(* CODESYS project elation_objectprog

Project tree, tasks and I/O mapping:
  Device : CODESYS Control for Linux SL, CODESYS, order no. 2302000005, version 4.13.0.0
    application Application
      libraries: Standard, 3.5.18.0 (System); Util, 3.5.19.0 (System); VisuDialogs, * (System)
      task MainTask (cyclic, interval t#4ms, priority 1) calls Main_program
      task VISU_TASK (cyclic, interval 100 ms, priority 31) calls VisuElems.Visu_Prg
      Chiller_funct/
        function maskbitFunction [ST]
        function scaleFunction [ST]
      function block clsLampFunction [ST]: Lamp, Switch, Value
      function block FB_Provision_room [ST]: MET_assign_values, P_Alarm, P_Defrost, P_Defrost_end_temperature, P_Door_open, P_Dout2, P_Dout3, P_Drain_down_time, P_Generic_alarm, P_High_temperature_alarm_threshold, P_High_temperature, P_Low_temperature, P_Low_temperature_alarm_threshold, P_Machine_standby, P_Maximum_defrost_duration, P_Provision_name, P_Room_temp, P_Setpoint, P_T1_failure, P_T2_failure, P_Temp_defrost, P_Thermostat_OFF_ON_ref_to_SP, P_Thermostat_ON_OFF_ref_to_SP, P_Time_based_defrost, MET_write_sepoint, P_setpoint_write, P_test_input, P_Thermostat_OFF_ON_ref_to_SP_write, P_Thermostat_ON_OFF_ref_to_SP_write, P_xTrigger_setpoint
      interface IProvroom: Lamp, Switch, Value
      interface ITF_provision_room: MET_assign_values, P_Alarm, P_Defrost, P_Defrost_end_temperature, P_Door_open, P_Dout2, P_Dout3, P_Drain_down_time, P_Generic_alarm, P_High_temperature, P_High_temperature_alarm_threshold, P_Low_temperature, P_Low_temperature_alarm_threshold, P_Machine_standby, P_Maximum_defrost_duration, P_Provision_name, P_Room_temp, P_Setpoint, P_T1_failure, P_T2_failure, P_Temp_defrost, P_Thermostat_OFF_ON_ref_to_SP, P_Thermostat_ON_OFF_ref_to_SP, P_Time_based_defrost, MET_write_sepoint, P_setpoint_write, P_test_input, P_Thermostat_OFF_ON_ref_to_SP_write, P_Thermostat_ON_OFF_ref_to_SP_write
      program Main_program [ST]
      visualisation MainVisualization
      visualisation objectvisiu
      visualisation Provision_1_2_3_SysOverview
      program Provision_1 [ST]
      visualisation Provision_1_Values
      program Provision_2 [ST]
      program Provision_3 [ST]
      program Provision_4 [ST]
      visualisation Provision_overview
      visualisation ProvRoom_All
      visualisation ProvRoomTemp
    Modbus_COM_2 : Modbus COM, CODESYS, version 4.4.0.0
        settings: ComPort = 2
      Modbus_Master_COM_Port : Modbus Client, COM Port, CODESYS, version 4.4.0.0
          settings: Auto-restart communication = TRUE
        Modbus_Slave_COM_Prov1 : Modbus Server, COM Port, CODESYS, version 4.4.0.0
            settings: Channel 0.Function Code = 3; Channel 0.Read Offset = 16#0000; Channel 0.Read Length = 18; Channel 0.Write Offset = 0; Channel 0.Write Length = 0; Channel 0.Cycle Time = 100; Channel 1.Function Code = 3; Channel 1.Read Offset = 16#0064; Channel 1.Read Length = 3; Channel 1.Write Offset = 0; Channel 1.Write Length = 0; Channel 1.Cycle Time = 100; Channel 2.Function Code = 3; Channel 2.Read Offset = 16#00C8; Channel 2.Read Length = 11; Channel 2.Write Offset = 0; Channel 2.Write Length = 0; Channel 2.Cycle Time = 100; Channel 3.Function Code = 3; Channel 3.Read Offset = 16#012C; Channel 3.Read Length = 10; Channel 3.Write Offset = 0; Channel 3.Write Length = 0; Channel 3.Cycle Time = 100; Channel 4.Function Code = 3; Channel 4.Read Offset = 16#0190; Channel 4.Read Length = 13; Channel 4.Write Offset = 0; Channel 4.Write Length = 0; Channel 4.Cycle Time = 100; Channel 5.Function Code = 3; Channel 5.Read Offset = 16#01F4; Channel 5.Read Length = 9; Channel 5.Write Offset = 0; Channel 5.Write Length = 0; Channel 5.Cycle Time = 100; Channel 6.Function Code = 3; Channel 6.Read Offset = 16#0258; Channel 6.Read Length = 10; Channel 6.Write Offset = 0;
              Channel 6.Write Length = 0; Channel 6.Cycle Time = 100; Channel 7.Function Code = 3; Channel 7.Read Offset = 16#02BE; Channel 7.Read Length = 2; Channel 7.Write Offset = 0; Channel 7.Write Length = 0; Channel 7.Cycle Time = 100; Channel 8.Function Code = 3; Channel 8.Read Offset = 16#01C2; Channel 8.Read Length = 8; Channel 8.Write Offset = 0; Channel 8.Write Length = 0; Channel 8.Cycle Time = 100; Channel 9.Function Code = 3; Channel 9.Read Offset = 16#00C1; Channel 9.Read Length = 5; Channel 9.Write Offset = 0; Channel 9.Write Length = 0; Channel 9.Cycle Time = 100; Channel 10.Function Code = 3; Channel 10.Read Offset = 16#028A; Channel 10.Read Length = 4; Channel 10.Write Offset = 0; Channel 10.Write Length = 0; Channel 10.Cycle Time = 100; Channel 11.Function Code = 6; Channel 11.Read Offset = 0; Channel 11.Read Length = 0; Channel 11.Write Offset = 16#012F; Channel 11.Write Length = 1; Channel 11.Cycle Time = 100; Channel 12.Function Code = 6; Channel 12.Read Offset = 0; Channel 12.Read Length = 0; Channel 12.Write Offset = 16#02BE; Channel 12.Write Length = 1; Channel 12.Cycle Time = 100; Channel 13.Function Code = 6; Channel 13.Read Offset = 0;
              Channel 13.Read Length = 0; Channel 13.Write Offset = 16#0130; Channel 13.Write Length = 1; Channel 13.Cycle Time = 100; Channel 14.Function Code = 6; Channel 14.Read Offset = 0; Channel 14.Read Length = 0; Channel 14.Write Offset = 16#0131; Channel 14.Write Length = 1; Channel 14.Cycle Time = 100; Channel 15.Function Code = 6; Channel 15.Read Offset = 0; Channel 15.Read Length = 0; Channel 15.Write Offset = 16#01F5; Channel 15.Write Length = 1; Channel 15.Cycle Time = 100; Channel 16.Function Code = 6; Channel 16.Read Offset = 0; Channel 16.Read Length = 0; Channel 16.Write Offset = 16#01F6; Channel 16.Write Length = 1; Channel 16.Cycle Time = 100; Channel 17.Function Code = 6; Channel 17.Read Offset = 0; Channel 17.Read Length = 0; Channel 17.Write Offset = 16#0079; Channel 17.Write Length = 1; Channel 17.Cycle Time = 100; Channel 18.Function Code = 6; Channel 18.Read Offset = 0; Channel 18.Read Length = 0; Channel 18.Write Offset = 16#0080; Channel 18.Write Length = 1; Channel 18.Cycle Time = 100; Channel 19.Function Code = 6; Channel 19.Read Offset = 0; Channel 19.Read Length = 0; Channel 19.Write Offset = 16#0191; Channel 19.Write Length = 1; Channel 19.Cycle Time = 100;
              Channel 20.Function Code = 6; Channel 20.Read Offset = 0; Channel 20.Read Length = 0; Channel 20.Write Offset = 16#0196; Channel 20.Write Length = 1; Channel 20.Cycle Time = 100; Channel 21.Function Code = 6; Channel 21.Read Offset = 0; Channel 21.Read Length = 0; Channel 21.Write Offset = 16#0198; Channel 21.Write Length = 1; Channel 21.Cycle Time = 100; Channel 22.Function Code = 6; Channel 22.Read Offset = 0; Channel 22.Read Length = 0; Channel 22.Write Offset = 16#0197; Channel 22.Write Length = 1; Channel 22.Cycle Time = 100; Channel 23.Function Code = 6; Channel 23.Read Offset = 0; Channel 23.Read Length = 0; Channel 23.Write Offset = 16#007A; Channel 23.Write Length = 1; Channel 23.Cycle Time = 100; Channel 24.Function Code = 6; Channel 24.Read Offset = 0; Channel 24.Read Length = 0; Channel 24.Write Offset = 16#01C2; Channel 24.Write Length = 1; Channel 24.Cycle Time = 100; Channel 25.Function Code = 6; Channel 25.Read Offset = 0; Channel 25.Read Length = 0; Channel 25.Write Offset = 16#00C8; Channel 25.Write Length = 1; Channel 25.Cycle Time = 100; Channel 26.Function Code = 6; Channel 26.Read Offset = 0; Channel 26.Read Length = 0; Channel 26.Write Offset = 16#012C;
              Channel 26.Write Length = 1; Channel 26.Cycle Time = 100; Channel 27.Function Code = 6; Channel 27.Read Offset = 0; Channel 27.Read Length = 0; Channel 27.Write Offset = 16#012D; Channel 27.Write Length = 1; Channel 27.Cycle Time = 100; Channel 28.Function Code = 6; Channel 28.Read Offset = 0; Channel 28.Read Length = 0; Channel 28.Write Offset = 16#012E; Channel 28.Write Length = 1; Channel 28.Cycle Time = 100; Channel 29.Function Code = 6; Channel 29.Read Offset = 0; Channel 29.Read Length = 0; Channel 29.Write Offset = 16#0132; Channel 29.Write Length = 1; Channel 29.Cycle Time = 100; Channel 30.Function Code = 6; Channel 30.Read Offset = 0; Channel 30.Read Length = 0; Channel 30.Write Offset = 16#0133; Channel 30.Write Length = 1; Channel 30.Cycle Time = 100; Channel 31.Function Code = 6; Channel 31.Read Offset = 0; Channel 31.Read Length = 0; Channel 31.Write Offset = 16#0134; Channel 31.Write Length = 1; Channel 31.Cycle Time = 100; Channel 32.Function Code = 6; Channel 32.Read Offset = 0; Channel 32.Read Length = 0; Channel 32.Write Offset = 16#0135; Channel 32.Write Length = 1; Channel 32.Cycle Time = 100; Channel 33.Function Code = 6; Channel 33.Read Offset = 0;
              Channel 33.Read Length = 0; Channel 33.Write Offset = 16#0192; Channel 33.Write Length = 1; Channel 33.Cycle Time = 100; Channel 34.Function Code = 6; Channel 34.Read Offset = 0; Channel 34.Read Length = 0; Channel 34.Write Offset = 16#0194; Channel 34.Write Length = 1; Channel 34.Cycle Time = 100; Channel 35.Function Code = 6; Channel 35.Read Offset = 0; Channel 35.Read Length = 0; Channel 35.Write Offset = 16#019C; Channel 35.Write Length = 1; Channel 35.Cycle Time = 100; Channel 36.Function Code = 6; Channel 36.Read Offset = 0; Channel 36.Read Length = 0; Channel 36.Write Offset = 16#019A; Channel 36.Write Length = 1; Channel 36.Cycle Time = 100; Channel 37.Function Code = 6; Channel 37.Read Offset = 0; Channel 37.Read Length = 0; Channel 37.Write Offset = 16#019B; Channel 37.Write Length = 1; Channel 37.Cycle Time = 100; Channel 45.Function Code = 6; Channel 45.Read Offset = 0; Channel 45.Read Length = 0; Channel 45.Write Offset = 16#01F4; Channel 45.Write Length = 1; Channel 45.Cycle Time = 100; Channel 39.Function Code = 6; Channel 39.Read Offset = 0; Channel 39.Read Length = 0; Channel 39.Write Offset = 16#01C3; Channel 39.Write Length = 1; Channel 39.Cycle Time = 100;
              Channel 40.Function Code = 6; Channel 40.Read Offset = 0; Channel 40.Read Length = 0; Channel 40.Write Offset = 16#01C4; Channel 40.Write Length = 1; Channel 40.Cycle Time = 100; Channel 41.Function Code = 6; Channel 41.Read Offset = 0; Channel 41.Read Length = 0; Channel 41.Write Offset = 16#01FA; Channel 41.Write Length = 1; Channel 41.Cycle Time = 100; Channel 42.Function Code = 6; Channel 42.Read Offset = 0; Channel 42.Read Length = 0; Channel 42.Write Offset = 16#0259; Channel 42.Write Length = 1; Channel 42.Cycle Time = 100; Channel 43.Function Code = 6; Channel 43.Read Offset = 0; Channel 43.Read Length = 0; Channel 43.Write Offset = 16#025A; Channel 43.Write Length = 1; Channel 43.Cycle Time = 100; Channel 44.Function Code = 6; Channel 44.Read Offset = 0; Channel 44.Read Length = 0; Channel 44.Write Offset = 16#025B; Channel 44.Write Length = 1; Channel 44.Cycle Time = 100; Channel 46.Function Code = 6; Channel 46.Read Offset = 0; Channel 46.Read Length = 0; Channel 46.Write Offset = 16#01F4; Channel 46.Write Length = 1; Channel 46.Cycle Time = 100; Channel 47.Function Code = 6; Channel 47.Read Offset = 0; Channel 47.Read Length = 0; Channel 47.Write Offset = 16#00D0;
              Channel 47.Write Length = 1; Channel 47.Cycle Time = 100; Channel 48.Function Code = 6; Channel 48.Read Offset = 0; Channel 48.Read Length = 0; Channel 48.Write Offset = 16#028A; Channel 48.Write Length = 1; Channel 48.Cycle Time = 100; Channel 49.Function Code = 6; Channel 49.Read Offset = 0; Channel 49.Read Length = 0; Channel 49.Write Offset = 16#028B; Channel 49.Write Length = 1; Channel 49.Cycle Time = 100; Channel 50.Function Code = 6; Channel 50.Read Offset = 0; Channel 50.Read Length = 0; Channel 50.Write Offset = 16#028C; Channel 50.Write Length = 1; Channel 50.Cycle Time = 100; Channel 51.Function Code = 6; Channel 51.Read Offset = 0; Channel 51.Read Length = 0; Channel 51.Write Offset = 16#028D; Channel 51.Write Length = 1; Channel 51.Cycle Time = 100; Channel 52.Function Code = 6; Channel 52.Read Offset = 0; Channel 52.Read Length = 0; Channel 52.Write Offset = 16#025C; Channel 52.Write Length = 1; Channel 52.Cycle Time = 100; Channel 53.Function Code = 6; Channel 53.Read Offset = 0; Channel 53.Read Length = 0; Channel 53.Write Offset = 16#025D; Channel 53.Write Length = 1; Channel 53.Cycle Time = 100; Channel 54.Function Code = 6; Channel 54.Read Offset = 0;
              Channel 54.Read Length = 0; Channel 54.Write Offset = 16#025E; Channel 54.Write Length = 1; Channel 54.Cycle Time = 100; Channel 55.Function Code = 6; Channel 55.Read Offset = 0; Channel 55.Read Length = 0; Channel 55.Write Offset = 16#025F; Channel 55.Write Length = 1; Channel 55.Cycle Time = 100; Channel 56.Function Code = 6; Channel 56.Read Offset = 0; Channel 56.Read Length = 0; Channel 56.Write Offset = 16#0260; Channel 56.Write Length = 1; Channel 56.Cycle Time = 100; Channel 57.Function Code = 6; Channel 57.Read Offset = 0; Channel 57.Read Length = 0; Channel 57.Write Offset = 16#0261; Channel 57.Write Length = 1; Channel 57.Cycle Time = 100; Channel 58.Function Code = 6; Channel 58.Read Offset = 0; Channel 58.Read Length = 0; Channel 58.Write Offset = 16#0193; Channel 58.Write Length = 1; Channel 58.Cycle Time = 100
            input  Application.Main_program.modbus_var[1,0] : WORD  // Channel 0.Channel 0
            input  Application.Main_program.modbus_var[1,1] : WORD  // Channel 0.Channel 0
            input  Application.Main_program.modbus_var[1,2] : WORD  // Channel 0.Channel 0
            input  Application.Main_program.modbus_var[1,3] : WORD  // Channel 0.Channel 0
            input  Application.Main_program.modbus_var[1,4] : WORD  // Channel 0.Channel 0
            input  Application.Main_program.modbus_var[1,5] : WORD  // Channel 0.Channel 0
            input  Application.Main_program.modbus_var[1,6] : WORD  // Channel 0.Channel 0
            input  Application.Main_program.modbus_var[1,7] : WORD  // Channel 0.Channel 0
            input  Application.Main_program.modbus_var[1,8] : WORD  // Channel 0.Channel 0
            input  Application.Main_program.modbus_var[1,9] : WORD  // Channel 0.Channel 0
            input  Application.Main_program.modbus_var[1,10] : WORD  // Channel 0.Channel 0
            input  Application.Main_program.modbus_var[1,11] : WORD  // Channel 0.Channel 0
            input  Application.Main_program.modbus_var[1,12] : WORD  // Channel 0.Channel 0
            input  Application.Main_program.modbus_var[1,13] : WORD  // Channel 0.Channel 0
            input  Application.Main_program.modbus_var[1,14] : WORD  // Channel 0.Channel 0
            input  Application.Main_program.modbus_var[1,15] : WORD  // Channel 0.Channel 0
            input  Application.Main_program.modbus_var[1,16] : WORD  // Channel 0.Channel 0
            input  Application.Main_program.modbus_var[1,17] : WORD  // Channel 0.Channel 0
            input  Application.Main_program.modbus_var[1,100] : WORD  // Channel 1.Channel 1
            input  Application.Main_program.modbus_var[1,101] : WORD  // Channel 1.Channel 1
            input  Application.Main_program.modbus_var[1,102] : WORD  // Channel 1.Channel 1
            output Application.Provision_1.get_param_trigger.Q : BIT  // Channel 2
            input  Application.Main_program.modbus_var[1,200] : WORD  // Channel 2.Channel 2
            input  Application.Main_program.modbus_var[1,201] : WORD  // Channel 2.Channel 2
            input  Application.Main_program.modbus_var[1,202] : WORD  // Channel 2.Channel 2
            input  Application.Main_program.modbus_var[1,203] : WORD  // Channel 2.Channel 2
            input  Application.Main_program.modbus_var[1,204] : WORD  // Channel 2.Channel 2
            input  Application.Main_program.modbus_var[1,205] : WORD  // Channel 2.Channel 2
            input  Application.Main_program.modbus_var[1,206] : WORD  // Channel 2.Channel 2
            input  Application.Main_program.modbus_var[1,207] : WORD  // Channel 2.Channel 2
            input  Application.Main_program.modbus_var[1,208] : WORD  // Channel 2.Channel 2
            input  Application.Main_program.modbus_var[1,209] : WORD  // Channel 2.Channel 2
            input  Application.Main_program.modbus_var[1,210] : WORD  // Channel 2.Channel 2
            input  Application.Main_program.modbus_var[1,300] : WORD  // Channel 3.Channel 3
            input  Application.Main_program.modbus_var[1,301] : WORD  // Channel 3.Channel 3
            input  Application.Main_program.modbus_var[1,302] : WORD  // Channel 3.Channel 3
            input  Application.Main_program.modbus_var[1,303] : WORD  // Channel 3.Channel 3
            input  Application.Main_program.modbus_var[1,304] : WORD  // Channel 3.Channel 3
            input  Application.Main_program.modbus_var[1,305] : WORD  // Channel 3.Channel 3
            input  Application.Main_program.modbus_var[1,306] : WORD  // Channel 3.Channel 3
            input  Application.Main_program.modbus_var[1,307] : WORD  // Channel 3.Channel 3
            input  Application.Main_program.modbus_var[1,308] : WORD  // Channel 3.Channel 3
            input  Application.Main_program.modbus_var[1,309] : WORD  // Channel 3.Channel 3
            input  Application.Main_program.modbus_var[1,400] : WORD  // Channel 4.Channel 4
            input  Application.Main_program.modbus_var[1,401] : WORD  // Channel 4.Channel 4
            input  Application.Main_program.modbus_var[1,402] : WORD  // Channel 4.Channel 4
            input  Application.Main_program.modbus_var[1,403] : WORD  // Channel 4.Channel 4
            input  Application.Main_program.modbus_var[1,404] : WORD  // Channel 4.Channel 4
            input  Application.Main_program.modbus_var[1,405] : WORD  // Channel 4.Channel 4
            input  Application.Main_program.modbus_var[1,406] : WORD  // Channel 4.Channel 4
            input  Application.Main_program.modbus_var[1,407] : WORD  // Channel 4.Channel 4
            input  Application.Main_program.modbus_var[1,408] : WORD  // Channel 4.Channel 4
            input  Application.Main_program.modbus_var[1,409] : WORD  // Channel 4.Channel 4
            input  Application.Main_program.modbus_var[1,410] : WORD  // Channel 4.Channel 4
            input  Application.Main_program.modbus_var[1,411] : WORD  // Channel 4.Channel 4
            input  Application.Main_program.modbus_var[1,412] : WORD  // Channel 4.Channel 4
            input  Application.Main_program.modbus_var[1,500] : WORD  // Channel 5.Channel 5
            input  Application.Main_program.modbus_var[1,501] : WORD  // Channel 5.Channel 5
            input  Application.Main_program.modbus_var[1,502] : WORD  // Channel 5.Channel 5
            input  Application.Main_program.modbus_var[1,503] : WORD  // Channel 5.Channel 5
            input  Application.Main_program.modbus_var[1,504] : WORD  // Channel 5.Channel 5
            input  Application.Main_program.modbus_var[1,505] : WORD  // Channel 5.Channel 5
            input  Application.Main_program.modbus_var[1,506] : WORD  // Channel 5.Channel 5
            input  Application.Main_program.modbus_var[1,507] : WORD  // Channel 5.Channel 5
            input  Application.Main_program.modbus_var[1,508] : WORD  // Channel 5.Channel 5
            output Application.Provision_1.get_param_trigger.Q : BIT  // Channel 6
            input  Application.Main_program.modbus_var[1,600] : WORD  // Channel 6.Channel 6
            input  Application.Main_program.modbus_var[1,601] : WORD  // Channel 6.Channel 6
            input  Application.Main_program.modbus_var[1,602] : WORD  // Channel 6.Channel 6
            input  Application.Main_program.modbus_var[1,603] : WORD  // Channel 6.Channel 6
            input  Application.Main_program.modbus_var[1,604] : WORD  // Channel 6.Channel 6
            input  Application.Main_program.modbus_var[1,605] : WORD  // Channel 6.Channel 6
            input  Application.Main_program.modbus_var[1,606] : WORD  // Channel 6.Channel 6
            input  Application.Main_program.modbus_var[1,607] : WORD  // Channel 6.Channel 6
            input  Application.Main_program.modbus_var[1,608] : WORD  // Channel 6.Channel 6
            input  Application.Main_program.modbus_var[1,609] : WORD  // Channel 6.Channel 6
            output Application.Provision_1.get_param_trigger.Q : BIT  // Channel 7
            input  Application.Main_program.modbus_var[1,702] : WORD  // Channel 7.Channel 7
            input  Application.Main_program.modbus_var[1,703] : WORD  // Channel 7.Channel 7
            output Application.Provision_1.get_param_trigger.Q : BIT  // Channel 8
            input  Application.Main_program.modbus_var[1,450] : WORD  // Channel 8.Channel 8
            input  Application.Main_program.modbus_var[1,451] : WORD  // Channel 8.Channel 8
            input  Application.Main_program.modbus_var[1,452] : WORD  // Channel 8.Channel 8
            input  Application.Main_program.modbus_var[1,453] : WORD  // Channel 8.Channel 8
            input  Application.Main_program.modbus_var[1,454] : WORD  // Channel 8.Channel 8
            input  Application.Main_program.modbus_var[1,455] : WORD  // Channel 8.Channel 8
            input  Application.Main_program.modbus_var[1,456] : WORD  // Channel 8.Channel 8
            input  Application.Main_program.modbus_var[1,457] : WORD  // Channel 8.Channel 8
            output Application.Provision_1.get_param_trigger.Q : BIT  // Channel 9
            output Application.Provision_1.get_param_trigger.Q : BIT  // Channel 10
            input  Application.Main_program.modbus_var[1,650] : WORD  // Channel 10.Channel 10
            input  Application.Main_program.modbus_var[1,651] : WORD  // Channel 10.Channel 10
            input  Application.Main_program.modbus_var[1,652] : WORD  // Channel 10.Channel 10
            input  Application.Main_program.modbus_var[1,653] : WORD  // Channel 10.Channel 10
            output Application.Provision_1.write_data_setp.Q : BIT  // Channel 11
            output Application.Provision_1.setp_write_word : WORD  // Channel 11.Channel 11
            output Application.Provision_1.write_data_control.Q : BIT  // Channel 12
            output Application.Provision_1.standby_write : WORD  // Channel 12.Channel 12
            output Application.Provision_1.write_data_setp.Q : BIT  // Channel 13
            output Application.Provision_1.Thermostat_OFF_ON_write_word : WORD  // Channel 13.Channel 13
            output Application.Provision_1.write_data_setp.Q : BIT  // Channel 14
            output Application.Provision_1.Thermostat_ON_OFF_write_word : WORD  // Channel 14.Channel 14
            output Application.Provision_1.write_data_alarm.Q : BIT  // Channel 15
            output Application.Provision_1.Low_temperature_alarm_thres_write_word : WORD  // Channel 15.Channel 15
            output Application.Provision_1.write_data_alarm.Q : BIT  // Channel 16
            output Application.Provision_1.High_temperature_alarm_thres_write_word : WORD  // Channel 16.Channel 16
            output Application.Provision_1.write_data_mute.Q : BIT  // Channel 17
            output Application.Provision_1.muteAlarm : WORD  // Channel 17.Channel 17
            output Application.Provision_1.Time_based_defrost_write_word : WORD  // Channel 18.Channel 18
            output Application.Provision_1.write_data_defrost.Q : BIT  // Channel 19
            output Application.Provision_1.Time_based_defrost_write_word : WORD  // Channel 19.Channel 19
            output Application.Provision_1.write_data_defrost.Q : BIT  // Channel 20
            output Application.Provision_1.Defrost_end_temperature_write_word : WORD  // Channel 20.Channel 20
            output Application.Provision_1.write_data_defrost.Q : BIT  // Channel 21
            output Application.Provision_1.Drain_down_time_write_int : WORD  // Channel 21.Channel 21
            output Application.Provision_1.write_data_defrost.Q : BIT  // Channel 22
            output Application.Provision_1.Maximum_defrost_duration_write_word : WORD  // Channel 22.Channel 22
            output Application.Provision_1.write_data_man_defrost.Q : BIT  // Channel 23
            output Application.Provision_1.defrost_write : WORD  // Channel 23.Channel 23
            output Application.Provision_1.set_param_trigger.Q : BIT  // Channel 24
            output Application.Provision_1.Fan_stop_temperature_write_word : WORD  // Channel 24.Channel 24
            output Application.Provision_1.preset_parameters_write_int : WORD  // Channel 25.Channel 25
            output Application.Provision_1.set_param_trigger.Q : BIT  // Channel 26
            output Application.Provision_1.Readout_scale_write_int : WORD  // Channel 26.Channel 26
            output Application.Provision_1.set_param_trigger.Q : BIT  // Channel 27
            output Application.Provision_1.Minimum_temperature_setpoint_write_int : WORD  // Channel 27.Channel 27
            output Application.Provision_1.set_param_trigger.Q : BIT  // Channel 28
            output Application.Provision_1.Maximum_temperature_setpoint_write_int : WORD  // Channel 28.Channel 28
            output Application.Provision_1.set_param_trigger.Q : BIT  // Channel 29
            output Application.Provision_1.CH_minimum_OFF_time_write_int : WORD  // Channel 29.Channel 29
            output Application.Provision_1.set_param_trigger.Q : BIT  // Channel 30
            output Application.Provision_1.CH_minimum_ON_time_write_int : WORD  // Channel 30.Channel 30
            output Application.Provision_1.set_param_trigger.Q : BIT  // Channel 31
            output Application.Provision_1.CH_output_ON_when_probe_T1_is_faulty_write_int : WORD  // Channel 31.Channel 31
            output Application.Provision_1.set_param_trigger.Q : BIT  // Channel 32
            output Application.Provision_1.CH_output_OFF_when_probe_T1_is_faulty_write_int : WORD  // Channel 32.Channel 32
            output Application.Provision_1.set_param_trigger.Q : BIT  // Channel 33
            output Application.Provision_1.Minimum_Time_Between_Defrost_write_int : WORD  // Channel 33.Channel 33
            output Application.Provision_1.set_param_trigger.Q : BIT  // Channel 34
            output Application.Provision_1.Defrost_type_write_int : WORD  // Channel 34.Channel 34
            output Application.Provision_1.set_param_trigger.Q : BIT  // Channel 35
            output Application.Provision_1.Fan_restart_temperature_after_defrost_write_int : WORD  // Channel 35.Channel 35
            output Application.Provision_1.set_param_trigger.Q : BIT  // Channel 36
            output Application.Provision_1.Display_delay_write_int : WORD  // Channel 36.Channel 36
            output Application.Provision_1.set_param_trigger.Q : BIT  // Channel 37
            output Application.Provision_1.Fans_active_during_defrost_write_int : WORD  // Channel 37.Channel 37
            output Application.Provision_1.set_param_trigger.Q : BIT  // Channel 39
            output Application.Provision_1.Maximum_fan_stop_for_FDD_FET_write_int : WORD  // Channel 39.Channel 39
            output Application.Provision_1.set_param_trigger.Q : BIT  // Channel 40
            output Application.Provision_1.Fan_mode_during_thermostatic_control_write_int : WORD  // Channel 40.Channel 40
            output Application.Provision_1.set_param_trigger.Q : BIT  // Channel 41
            output Application.Provision_1.Temperature_alarm_delay_write_int : WORD  // Channel 41.Channel 41
            output Application.Provision_1.set_param_trigger.Q : BIT  // Channel 42
            output Application.Provision_1.Door_switch_input_mode_write_int : WORD  // Channel 42.Channel 42
            output Application.Provision_1.set_param_trigger.Q : BIT  // Channel 43
            output Application.Provision_1.Door_alarm_delay_write_int : WORD  // Channel 43.Channel 43
            output Application.Provision_1.set_param_trigger.Q : BIT  // Channel 44
            output Application.Provision_1.Compressor_stop_delay_write_int : WORD  // Channel 44.Channel 44
            output Application.Provision_1.set_param_trigger.Q : BIT  // Channel 46
            output Application.Provision_1.Alarm_threshold_management_write_int : WORD  // Channel 46.Channel 46
            output Application.Provision_1.set_param_trigger.Q : BIT  // Channel 47
            output Application.Provision_1.Display_slowdown_write_int : WORD  // Channel 47.Channel 47
            output Application.Provision_1.set_param_trigger.Q : BIT  // Channel 48
            output Application.Provision_1.RL1_output_operation_write_int : WORD  // Channel 48.Channel 48
            output Application.Provision_1.set_param_trigger.Q : BIT  // Channel 49
            output Application.Provision_1.RL2_output_operation_write_int : WORD  // Channel 49.Channel 49
            output Application.Provision_1.set_param_trigger.Q : BIT  // Channel 50
            output Application.Provision_1.RL3_output_operation_write_int : WORD  // Channel 50.Channel 50
            output Application.Provision_1.set_param_trigger.Q : BIT  // Channel 51
            output Application.Provision_1.RL4_output_operation_write_int : WORD  // Channel 51.Channel 51
            output Application.Provision_1.Door_stop_timeout_write_int : WORD  // Channel 52.Channel 52
            output Application.Provision_1.set_param_trigger.Q : BIT  // Channel 53
            output Application.Provision_1.DI1_digital_input_operation_write_int : WORD  // Channel 53.Channel 53
            output Application.Provision_1.set_param_trigger.Q : BIT  // Channel 54
            output Application.Provision_1.DI1_digital_input_activation_write_int : WORD  // Channel 54.Channel 54
            output Application.Provision_1.set_param_trigger.Q : BIT  // Channel 55
            output Application.Provision_1.DI2_digital_input_operation_write_int : WORD  // Channel 55.Channel 55
            output Application.Provision_1.set_param_trigger.Q : BIT  // Channel 56
            output Application.Provision_1.DI2_digital_input_activation_write_int : WORD  // Channel 56.Channel 56
            output Application.Provision_1.set_param_trigger.Q : BIT  // Channel 57
            output Application.Provision_1.Light_control_mode_write_int : WORD  // Channel 57.Channel 57
            output Application.Provision_1.set_param_trigger.Q : BIT  // Channel 58
            output Application.Provision_1.Defrost_time_optimization_write_int : WORD  // Channel 58.Channel 58
            unmapped channels: Channel 0, Channel 1, Channel 2, Channel 3, Channel 4, Channel 5, Channel 6, Channel 7, Channel 8, Channel 9, Channel 10, Channel 11, Channel 12, Channel 13, Channel 14, Channel 15, Channel 16, Channel 17, Channel 18, Channel 18, Channel 19, Channel 20, Channel 21, Channel 22, Channel 23, Channel 24, Channel 25, Channel 25, Channel 26, Channel 27, Channel 28, Channel 29, Channel 30, Channel 31, Channel 32, Channel 33, Channel 34, Channel 35, Channel 36, Channel 37,
              Channel 38, Channel 45, Channel 39, Channel 40, Channel 41, Channel 42, Channel 43, Channel 44, Channel 46, Channel 47, Channel 48, Channel 49, Channel 50, Channel 51, Channel 52, Channel 53, Channel 54, Channel 55, Channel 56, Channel 57, Channel 58
        Modbus_Slave_COM_Prov2 : Modbus Server, COM Port, CODESYS, version 4.4.0.0
            settings: SlaveAddress = 2; ResponseTimeout = 1000; UseExtendedFunctionCodes = TRUE; Channel 0.Function Code = 3; Channel 0.Read Offset = 16#0000; Channel 0.Read Length = 18; Channel 0.Write Offset = 0; Channel 0.Write Length = 0; Channel 0.Cycle Time = 100; Channel 1.Function Code = 3; Channel 1.Read Offset = 16#0064; Channel 1.Read Length = 3; Channel 1.Write Offset = 0; Channel 1.Write Length = 0; Channel 1.Cycle Time = 100; Channel 2.Function Code = 3; Channel 2.Read Offset = 16#00C8; Channel 2.Read Length = 11; Channel 2.Write Offset = 0; Channel 2.Write Length = 0; Channel 2.Cycle Time = 100; Channel 3.Function Code = 3; Channel 3.Read Offset = 16#012C; Channel 3.Read Length = 10; Channel 3.Write Offset = 0; Channel 3.Write Length = 0; Channel 3.Cycle Time = 100; Channel 4.Function Code = 3; Channel 4.Read Offset = 16#0190; Channel 4.Read Length = 13; Channel 4.Write Offset = 0; Channel 4.Write Length = 0; Channel 4.Cycle Time = 100; Channel 5.Function Code = 3; Channel 5.Read Offset = 16#01F4; Channel 5.Read Length = 9; Channel 5.Write Offset = 0; Channel 5.Write Length = 0; Channel 5.Cycle Time = 100; Channel 6.Function Code = 3;
              Channel 6.Read Offset = 16#0258; Channel 6.Read Length = 10; Channel 6.Write Offset = 0; Channel 6.Write Length = 0; Channel 6.Cycle Time = 100; Channel 7.Function Code = 3; Channel 7.Read Offset = 16#02BE; Channel 7.Read Length = 2; Channel 7.Write Offset = 0; Channel 7.Write Length = 0; Channel 7.Cycle Time = 100; Channel 8.Function Code = 3; Channel 8.Read Offset = 16#01C2; Channel 8.Read Length = 8; Channel 8.Write Offset = 0; Channel 8.Write Length = 0; Channel 8.Cycle Time = 100; Channel 9.Function Code = 3; Channel 9.Read Offset = 16#00C1; Channel 9.Read Length = 5; Channel 9.Write Offset = 0; Channel 9.Write Length = 0; Channel 9.Cycle Time = 100; Channel 10.Function Code = 3; Channel 10.Read Offset = 16#028A; Channel 10.Read Length = 4; Channel 10.Write Offset = 0; Channel 10.Write Length = 0; Channel 10.Cycle Time = 100; Channel 11.Function Code = 6; Channel 11.Read Offset = 0; Channel 11.Read Length = 0; Channel 11.Write Offset = 16#012F; Channel 11.Write Length = 1; Channel 11.Cycle Time = 100; Channel 12.Function Code = 6; Channel 12.Read Offset = 0; Channel 12.Read Length = 0; Channel 12.Write Offset = 16#02BE; Channel 12.Write Length = 1;
              Channel 12.Cycle Time = 100; Channel 13.Function Code = 6; Channel 13.Read Offset = 0; Channel 13.Read Length = 0; Channel 13.Write Offset = 16#0130; Channel 13.Write Length = 1; Channel 13.Cycle Time = 100; Channel 14.Function Code = 6; Channel 14.Read Offset = 0; Channel 14.Read Length = 0; Channel 14.Write Offset = 16#0131; Channel 14.Write Length = 1; Channel 14.Cycle Time = 100; Channel 15.Function Code = 6; Channel 15.Read Offset = 0; Channel 15.Read Length = 0; Channel 15.Write Offset = 16#01F5; Channel 15.Write Length = 1; Channel 15.Cycle Time = 100; Channel 16.Function Code = 6; Channel 16.Read Offset = 0; Channel 16.Read Length = 0; Channel 16.Write Offset = 16#01F6; Channel 16.Write Length = 1; Channel 16.Cycle Time = 100; Channel 17.Function Code = 6; Channel 17.Read Offset = 0; Channel 17.Read Length = 0; Channel 17.Write Offset = 16#0079; Channel 17.Write Length = 1; Channel 17.Cycle Time = 100; Channel 18.Function Code = 6; Channel 18.Read Offset = 0; Channel 18.Read Length = 0; Channel 18.Write Offset = 16#0080; Channel 18.Write Length = 1; Channel 18.Cycle Time = 100; Channel 19.Function Code = 6; Channel 19.Read Offset = 0; Channel 19.Read Length = 0;
              Channel 19.Write Offset = 16#0191; Channel 19.Write Length = 1; Channel 19.Cycle Time = 100; Channel 20.Function Code = 6; Channel 20.Read Offset = 0; Channel 20.Read Length = 0; Channel 20.Write Offset = 16#0196; Channel 20.Write Length = 1; Channel 20.Cycle Time = 100; Channel 21.Function Code = 6; Channel 21.Read Offset = 0; Channel 21.Read Length = 0; Channel 21.Write Offset = 16#0198; Channel 21.Write Length = 1; Channel 21.Cycle Time = 100; Channel 22.Function Code = 6; Channel 22.Read Offset = 0; Channel 22.Read Length = 0; Channel 22.Write Offset = 16#0197; Channel 22.Write Length = 1; Channel 22.Cycle Time = 100; Channel 23.Function Code = 6; Channel 23.Read Offset = 0; Channel 23.Read Length = 0; Channel 23.Write Offset = 16#007A; Channel 23.Write Length = 1; Channel 23.Cycle Time = 100; Channel 24.Function Code = 6; Channel 24.Read Offset = 0; Channel 24.Read Length = 0; Channel 24.Write Offset = 16#01C2; Channel 24.Write Length = 1; Channel 24.Cycle Time = 100; Channel 25.Function Code = 6; Channel 25.Read Offset = 0; Channel 25.Read Length = 0; Channel 25.Write Offset = 16#00C8; Channel 25.Write Length = 1; Channel 25.Cycle Time = 100; Channel 26.Function Code = 6;
              Channel 26.Read Offset = 0; Channel 26.Read Length = 0; Channel 26.Write Offset = 16#012C; Channel 26.Write Length = 1; Channel 26.Cycle Time = 100; Channel 27.Function Code = 6; Channel 27.Read Offset = 0; Channel 27.Read Length = 0; Channel 27.Write Offset = 16#012D; Channel 27.Write Length = 1; Channel 27.Cycle Time = 100; Channel 28.Function Code = 6; Channel 28.Read Offset = 0; Channel 28.Read Length = 0; Channel 28.Write Offset = 16#012E; Channel 28.Write Length = 1; Channel 28.Cycle Time = 100; Channel 29.Function Code = 6; Channel 29.Read Offset = 0; Channel 29.Read Length = 0; Channel 29.Write Offset = 16#0132; Channel 29.Write Length = 1; Channel 29.Cycle Time = 100; Channel 30.Function Code = 6; Channel 30.Read Offset = 0; Channel 30.Read Length = 0; Channel 30.Write Offset = 16#0133; Channel 30.Write Length = 1; Channel 30.Cycle Time = 100; Channel 31.Function Code = 6; Channel 31.Read Offset = 0; Channel 31.Read Length = 0; Channel 31.Write Offset = 16#0134; Channel 31.Write Length = 1; Channel 31.Cycle Time = 100; Channel 32.Function Code = 6; Channel 32.Read Offset = 0; Channel 32.Read Length = 0; Channel 32.Write Offset = 16#0135; Channel 32.Write Length = 1;
              Channel 32.Cycle Time = 100; Channel 33.Function Code = 6; Channel 33.Read Offset = 0; Channel 33.Read Length = 0; Channel 33.Write Offset = 16#0192; Channel 33.Write Length = 1; Channel 33.Cycle Time = 100; Channel 34.Function Code = 6; Channel 34.Read Offset = 0; Channel 34.Read Length = 0; Channel 34.Write Offset = 16#0194; Channel 34.Write Length = 1; Channel 34.Cycle Time = 100; Channel 35.Function Code = 6; Channel 35.Read Offset = 0; Channel 35.Read Length = 0; Channel 35.Write Offset = 16#019C; Channel 35.Write Length = 1; Channel 35.Cycle Time = 100; Channel 36.Function Code = 6; Channel 36.Read Offset = 0; Channel 36.Read Length = 0; Channel 36.Write Offset = 16#019A; Channel 36.Write Length = 1; Channel 36.Cycle Time = 100; Channel 37.Function Code = 6; Channel 37.Read Offset = 0; Channel 37.Read Length = 0; Channel 37.Write Offset = 16#019B; Channel 37.Write Length = 1; Channel 37.Cycle Time = 100; Channel 45.Function Code = 6; Channel 45.Read Offset = 0; Channel 45.Read Length = 0; Channel 45.Write Offset = 16#01F4; Channel 45.Write Length = 1; Channel 45.Cycle Time = 100; Channel 39.Function Code = 6; Channel 39.Read Offset = 0; Channel 39.Read Length = 0;
              Channel 39.Write Offset = 16#01C3; Channel 39.Write Length = 1; Channel 39.Cycle Time = 100; Channel 40.Function Code = 6; Channel 40.Read Offset = 0; Channel 40.Read Length = 0; Channel 40.Write Offset = 16#01C4; Channel 40.Write Length = 1; Channel 40.Cycle Time = 100; Channel 41.Function Code = 6; Channel 41.Read Offset = 0; Channel 41.Read Length = 0; Channel 41.Write Offset = 16#01FA; Channel 41.Write Length = 1; Channel 41.Cycle Time = 100; Channel 42.Function Code = 6; Channel 42.Read Offset = 0; Channel 42.Read Length = 0; Channel 42.Write Offset = 16#0259; Channel 42.Write Length = 1; Channel 42.Cycle Time = 100; Channel 43.Function Code = 6; Channel 43.Read Offset = 0; Channel 43.Read Length = 0; Channel 43.Write Offset = 16#025A; Channel 43.Write Length = 1; Channel 43.Cycle Time = 100; Channel 44.Function Code = 6; Channel 44.Read Offset = 0; Channel 44.Read Length = 0; Channel 44.Write Offset = 16#025B; Channel 44.Write Length = 1; Channel 44.Cycle Time = 100; Channel 46.Function Code = 6; Channel 46.Read Offset = 0; Channel 46.Read Length = 0; Channel 46.Write Offset = 16#01F4; Channel 46.Write Length = 1; Channel 46.Cycle Time = 100; Channel 47.Function Code = 6;
              Channel 47.Read Offset = 0; Channel 47.Read Length = 0; Channel 47.Write Offset = 16#00D0; Channel 47.Write Length = 1; Channel 47.Cycle Time = 100; Channel 48.Function Code = 6; Channel 48.Read Offset = 0; Channel 48.Read Length = 0; Channel 48.Write Offset = 16#028A; Channel 48.Write Length = 1; Channel 48.Cycle Time = 100; Channel 49.Function Code = 6; Channel 49.Read Offset = 0; Channel 49.Read Length = 0; Channel 49.Write Offset = 16#028B; Channel 49.Write Length = 1; Channel 49.Cycle Time = 100; Channel 50.Function Code = 6; Channel 50.Read Offset = 0; Channel 50.Read Length = 0; Channel 50.Write Offset = 16#028C; Channel 50.Write Length = 1; Channel 50.Cycle Time = 100; Channel 51.Function Code = 6; Channel 51.Read Offset = 0; Channel 51.Read Length = 0; Channel 51.Write Offset = 16#028D; Channel 51.Write Length = 1; Channel 51.Cycle Time = 100; Channel 52.Function Code = 6; Channel 52.Read Offset = 0; Channel 52.Read Length = 0; Channel 52.Write Offset = 16#025C; Channel 52.Write Length = 1; Channel 52.Cycle Time = 100; Channel 53.Function Code = 6; Channel 53.Read Offset = 0; Channel 53.Read Length = 0; Channel 53.Write Offset = 16#025D; Channel 53.Write Length = 1;
              Channel 53.Cycle Time = 100; Channel 54.Function Code = 6; Channel 54.Read Offset = 0; Channel 54.Read Length = 0; Channel 54.Write Offset = 16#025E; Channel 54.Write Length = 1; Channel 54.Cycle Time = 100; Channel 55.Function Code = 6; Channel 55.Read Offset = 0; Channel 55.Read Length = 0; Channel 55.Write Offset = 16#025F; Channel 55.Write Length = 1; Channel 55.Cycle Time = 100; Channel 56.Function Code = 6; Channel 56.Read Offset = 0; Channel 56.Read Length = 0; Channel 56.Write Offset = 16#0260; Channel 56.Write Length = 1; Channel 56.Cycle Time = 100; Channel 57.Function Code = 6; Channel 57.Read Offset = 0; Channel 57.Read Length = 0; Channel 57.Write Offset = 16#0261; Channel 57.Write Length = 1; Channel 57.Cycle Time = 100; Channel 58.Function Code = 6; Channel 58.Read Offset = 0; Channel 58.Read Length = 0; Channel 58.Write Offset = 16#0193; Channel 58.Write Length = 1; Channel 58.Cycle Time = 100
            input  Application.Main_program.modbus_var[2,0] : WORD  // Channel 0.Channel 0
            input  Application.Main_program.modbus_var[2,1] : WORD  // Channel 0.Channel 0
            input  Application.Main_program.modbus_var[2,2] : WORD  // Channel 0.Channel 0
            input  Application.Main_program.modbus_var[2,3] : WORD  // Channel 0.Channel 0
            input  Application.Main_program.modbus_var[2,4] : WORD  // Channel 0.Channel 0
            input  Application.Main_program.modbus_var[2,5] : WORD  // Channel 0.Channel 0
            input  Application.Main_program.modbus_var[2,6] : WORD  // Channel 0.Channel 0
            input  Application.Main_program.modbus_var[2,7] : WORD  // Channel 0.Channel 0
            input  Application.Main_program.modbus_var[2,8] : WORD  // Channel 0.Channel 0
            input  Application.Main_program.modbus_var[2,9] : WORD  // Channel 0.Channel 0
            input  Application.Main_program.modbus_var[2,10] : WORD  // Channel 0.Channel 0
            input  Application.Main_program.modbus_var[2,11] : WORD  // Channel 0.Channel 0
            input  Application.Main_program.modbus_var[2,12] : WORD  // Channel 0.Channel 0
            input  Application.Main_program.modbus_var[2,13] : WORD  // Channel 0.Channel 0
            input  Application.Main_program.modbus_var[2,14] : WORD  // Channel 0.Channel 0
            input  Application.Main_program.modbus_var[2,15] : WORD  // Channel 0.Channel 0
            input  Application.Main_program.modbus_var[2,16] : WORD  // Channel 0.Channel 0
            input  Application.Main_program.modbus_var[2,17] : WORD  // Channel 0.Channel 0
            input  Application.Main_program.modbus_var[2,100] : WORD  // Channel 1.Channel 1
            input  Application.Main_program.modbus_var[2,101] : WORD  // Channel 1.Channel 1
            input  Application.Main_program.modbus_var[2,102] : WORD  // Channel 1.Channel 1
            output Application.Provision_2.get_param_trigger.Q : BIT  // Channel 2
            input  Application.Main_program.modbus_var[2,200] : WORD  // Channel 2.Channel 2
            input  Application.Main_program.modbus_var[2,201] : WORD  // Channel 2.Channel 2
            input  Application.Main_program.modbus_var[2,202] : WORD  // Channel 2.Channel 2
            input  Application.Main_program.modbus_var[2,203] : WORD  // Channel 2.Channel 2
            input  Application.Main_program.modbus_var[2,204] : WORD  // Channel 2.Channel 2
            input  Application.Main_program.modbus_var[2,205] : WORD  // Channel 2.Channel 2
            input  Application.Main_program.modbus_var[2,206] : WORD  // Channel 2.Channel 2
            input  Application.Main_program.modbus_var[2,207] : WORD  // Channel 2.Channel 2
            input  Application.Main_program.modbus_var[2,208] : WORD  // Channel 2.Channel 2
            input  Application.Main_program.modbus_var[2,209] : WORD  // Channel 2.Channel 2
            input  Application.Main_program.modbus_var[2,210] : WORD  // Channel 2.Channel 2
            input  Application.Main_program.modbus_var[2,300] : WORD  // Channel 3.Channel 3
            input  Application.Main_program.modbus_var[2,301] : WORD  // Channel 3.Channel 3
            input  Application.Main_program.modbus_var[2,302] : WORD  // Channel 3.Channel 3
            input  Application.Main_program.modbus_var[2,303] : WORD  // Channel 3.Channel 3
            input  Application.Main_program.modbus_var[2,304] : WORD  // Channel 3.Channel 3
            input  Application.Main_program.modbus_var[2,305] : WORD  // Channel 3.Channel 3
            input  Application.Main_program.modbus_var[2,306] : WORD  // Channel 3.Channel 3
            input  Application.Main_program.modbus_var[2,307] : WORD  // Channel 3.Channel 3
            input  Application.Main_program.modbus_var[2,308] : WORD  // Channel 3.Channel 3
            input  Application.Main_program.modbus_var[2,309] : WORD  // Channel 3.Channel 3
            input  Application.Main_program.modbus_var[2,400] : WORD  // Channel 4.Channel 4
            input  Application.Main_program.modbus_var[2,401] : WORD  // Channel 4.Channel 4
            input  Application.Main_program.modbus_var[2,402] : WORD  // Channel 4.Channel 4
            input  Application.Main_program.modbus_var[2,403] : WORD  // Channel 4.Channel 4
            input  Application.Main_program.modbus_var[2,404] : WORD  // Channel 4.Channel 4
            input  Application.Main_program.modbus_var[2,405] : WORD  // Channel 4.Channel 4
            input  Application.Main_program.modbus_var[2,406] : WORD  // Channel 4.Channel 4
            input  Application.Main_program.modbus_var[2,407] : WORD  // Channel 4.Channel 4
            input  Application.Main_program.modbus_var[2,408] : WORD  // Channel 4.Channel 4
            input  Application.Main_program.modbus_var[2,409] : WORD  // Channel 4.Channel 4
            input  Application.Main_program.modbus_var[2,410] : WORD  // Channel 4.Channel 4
            input  Application.Main_program.modbus_var[2,411] : WORD  // Channel 4.Channel 4
            input  Application.Main_program.modbus_var[2,412] : WORD  // Channel 4.Channel 4
            input  Application.Main_program.modbus_var[2,500] : WORD  // Channel 5.Channel 5
            input  Application.Main_program.modbus_var[2,501] : WORD  // Channel 5.Channel 5
            input  Application.Main_program.modbus_var[2,502] : WORD  // Channel 5.Channel 5
            input  Application.Main_program.modbus_var[2,503] : WORD  // Channel 5.Channel 5
            input  Application.Main_program.modbus_var[2,504] : WORD  // Channel 5.Channel 5
            input  Application.Main_program.modbus_var[2,505] : WORD  // Channel 5.Channel 5
            input  Application.Main_program.modbus_var[2,506] : WORD  // Channel 5.Channel 5
            input  Application.Main_program.modbus_var[2,507] : WORD  // Channel 5.Channel 5
            input  Application.Main_program.modbus_var[2,508] : WORD  // Channel 5.Channel 5
            output Application.Provision_2.get_param_trigger.Q : BIT  // Channel 6
            input  Application.Main_program.modbus_var[2,600] : WORD  // Channel 6.Channel 6
            input  Application.Main_program.modbus_var[2,601] : WORD  // Channel 6.Channel 6
            input  Application.Main_program.modbus_var[2,602] : WORD  // Channel 6.Channel 6
            input  Application.Main_program.modbus_var[2,603] : WORD  // Channel 6.Channel 6
            input  Application.Main_program.modbus_var[2,604] : WORD  // Channel 6.Channel 6
            input  Application.Main_program.modbus_var[2,605] : WORD  // Channel 6.Channel 6
            input  Application.Main_program.modbus_var[2,606] : WORD  // Channel 6.Channel 6
            input  Application.Main_program.modbus_var[2,607] : WORD  // Channel 6.Channel 6
            input  Application.Main_program.modbus_var[2,608] : WORD  // Channel 6.Channel 6
            input  Application.Main_program.modbus_var[2,609] : WORD  // Channel 6.Channel 6
            output Application.Provision_2.get_param_trigger.Q : BIT  // Channel 7
            input  Application.Main_program.modbus_var[2,702] : WORD  // Channel 7.Channel 7
            input  Application.Main_program.modbus_var[2,703] : WORD  // Channel 7.Channel 7
            output Application.Provision_2.get_param_trigger.Q : BIT  // Channel 8
            input  Application.Main_program.modbus_var[2,450] : WORD  // Channel 8.Channel 8
            input  Application.Main_program.modbus_var[2,451] : WORD  // Channel 8.Channel 8
            input  Application.Main_program.modbus_var[2,452] : WORD  // Channel 8.Channel 8
            input  Application.Main_program.modbus_var[2,453] : WORD  // Channel 8.Channel 8
            input  Application.Main_program.modbus_var[2,454] : WORD  // Channel 8.Channel 8
            input  Application.Main_program.modbus_var[2,455] : WORD  // Channel 8.Channel 8
            input  Application.Main_program.modbus_var[2,456] : WORD  // Channel 8.Channel 8
            input  Application.Main_program.modbus_var[2,457] : WORD  // Channel 8.Channel 8
            output Application.Provision_2.get_param_trigger.Q : BIT  // Channel 9
            output Application.Provision_2.get_param_trigger.Q : BIT  // Channel 10
            input  Application.Main_program.modbus_var[2,650] : WORD  // Channel 10.Channel 10
            input  Application.Main_program.modbus_var[2,651] : WORD  // Channel 10.Channel 10
            input  Application.Main_program.modbus_var[2,652] : WORD  // Channel 10.Channel 10
            input  Application.Main_program.modbus_var[2,653] : WORD  // Channel 10.Channel 10
            output Application.Main_program.Provision_room2.O_write_data_setp.Q : BIT  // Channel 11
            output Application.Main_program.Provision_room2.O_word_setpoint : WORD  // Channel 11.Channel 11
            output Application.Provision_2.write_data_control.Q : BIT  // Channel 12
            output Application.Provision_2.standby_write : WORD  // Channel 12.Channel 12
            output Application.Main_program.Provision_room2.O_write_data_setp.Q : BIT  // Channel 13
            output Application.Provision_2.Thermostat_OFF_ON_write_word : WORD  // Channel 13.Channel 13
            output Application.Main_program.Provision_room2.O_write_data_setp.Q : BIT  // Channel 14
            output Application.Provision_2.Thermostat_ON_OFF_write_word : WORD  // Channel 14.Channel 14
            output Application.Provision_2.write_data_alarm.Q : BIT  // Channel 15
            output Application.Provision_2.Low_temperature_alarm_thres_write_word : WORD  // Channel 15.Channel 15
            output Application.Provision_2.write_data_alarm.Q : BIT  // Channel 16
            output Application.Provision_2.High_temperature_alarm_thres_write_word : WORD  // Channel 16.Channel 16
            output Application.Provision_2.write_data_mute.Q : BIT  // Channel 17
            output Application.Provision_2.muteAlarm : WORD  // Channel 17.Channel 17
            output Application.Provision_2.Time_based_defrost_write_word : WORD  // Channel 18.Channel 18
            output Application.Provision_2.write_data_defrost.Q : BIT  // Channel 19
            output Application.Provision_2.Time_based_defrost_write_word : WORD  // Channel 19.Channel 19
            output Application.Provision_2.write_data_defrost.Q : BIT  // Channel 20
            output Application.Provision_2.Defrost_end_temperature_write_word : WORD  // Channel 20.Channel 20
            output Application.Provision_2.write_data_defrost.Q : BIT  // Channel 21
            output Application.Provision_2.Drain_down_time_write_int : WORD  // Channel 21.Channel 21
            output Application.Provision_2.write_data_defrost.Q : BIT  // Channel 22
            output Application.Provision_2.Maximum_defrost_duration_write_word : WORD  // Channel 22.Channel 22
            output Application.Provision_2.write_data_man_defrost.Q : BIT  // Channel 23
            output Application.Provision_2.defrost_write : WORD  // Channel 23.Channel 23
            output Application.Provision_2.set_param_trigger.Q : BIT  // Channel 24
            output Application.Provision_2.Fan_stop_temperature_write_word : WORD  // Channel 24.Channel 24
            output Application.Provision_2.preset_parameters_write_int : WORD  // Channel 25.Channel 25
            output Application.Provision_2.set_param_trigger.Q : BIT  // Channel 26
            output Application.Provision_2.Readout_scale_write_int : WORD  // Channel 26.Channel 26
            output Application.Provision_2.set_param_trigger.Q : BIT  // Channel 27
            output Application.Provision_2.Minimum_temperature_setpoint_write_int : WORD  // Channel 27.Channel 27
            output Application.Provision_2.set_param_trigger.Q : BIT  // Channel 28
            output Application.Provision_2.Maximum_temperature_setpoint_write_int : WORD  // Channel 28.Channel 28
            output Application.Provision_2.set_param_trigger.Q : BIT  // Channel 29
            output Application.Provision_2.CH_minimum_OFF_time_write_int : WORD  // Channel 29.Channel 29
            output Application.Provision_2.set_param_trigger.Q : BIT  // Channel 30
            output Application.Provision_2.CH_minimum_ON_time_write_int : WORD  // Channel 30.Channel 30
            output Application.Provision_2.set_param_trigger.Q : BIT  // Channel 31
            output Application.Provision_2.CH_output_ON_when_probe_T1_is_faulty_write_int : WORD  // Channel 31.Channel 31
            output Application.Provision_2.set_param_trigger.Q : BIT  // Channel 32
            output Application.Provision_2.CH_output_OFF_when_probe_T1_is_faulty_write_int : WORD  // Channel 32.Channel 32
            output Application.Provision_2.set_param_trigger.Q : BIT  // Channel 33
            output Application.Provision_2.Minimum_Time_Between_Defrost_write_int : WORD  // Channel 33.Channel 33
            output Application.Provision_2.set_param_trigger.Q : BIT  // Channel 34
            output Application.Provision_2.Defrost_type_write_int : WORD  // Channel 34.Channel 34
            output Application.Provision_2.set_param_trigger.Q : BIT  // Channel 35
            output Application.Provision_2.Fan_restart_temperature_after_defrost_write_int : WORD  // Channel 35.Channel 35
            output Application.Provision_2.set_param_trigger.Q : BIT  // Channel 36
            output Application.Provision_2.Display_delay_write_int : WORD  // Channel 36.Channel 36
            output Application.Provision_2.set_param_trigger.Q : BIT  // Channel 37
            output Application.Provision_2.Fans_active_during_defrost_write_int : WORD  // Channel 37.Channel 37
            output Application.Provision_2.set_param_trigger.Q : BIT  // Channel 39
            output Application.Provision_2.Maximum_fan_stop_for_FDD_FET_write_int : WORD  // Channel 39.Channel 39
            output Application.Provision_2.set_param_trigger.Q : BIT  // Channel 40
            output Application.Provision_2.Fan_mode_during_thermostatic_control_write_int : WORD  // Channel 40.Channel 40
            output Application.Provision_2.set_param_trigger.Q : BIT  // Channel 41
            output Application.Provision_2.Temperature_alarm_delay_write_int : WORD  // Channel 41.Channel 41
            output Application.Provision_2.set_param_trigger.Q : BIT  // Channel 42
            output Application.Provision_2.Door_switch_input_mode_write_int : WORD  // Channel 42.Channel 42
            output Application.Provision_2.set_param_trigger.Q : BIT  // Channel 43
            output Application.Provision_2.Door_alarm_delay_write_int : WORD  // Channel 43.Channel 43
            output Application.Provision_2.set_param_trigger.Q : BIT  // Channel 44
            output Application.Provision_2.Compressor_stop_delay_write_int : WORD  // Channel 44.Channel 44
            output Application.Provision_2.set_param_trigger.Q : BIT  // Channel 46
            output Application.Provision_2.Alarm_threshold_management_write_int : WORD  // Channel 46.Channel 46
            output Application.Provision_2.set_param_trigger.Q : BIT  // Channel 47
            output Application.Provision_2.Display_slowdown_write_int : WORD  // Channel 47.Channel 47
            output Application.Provision_2.set_param_trigger.Q : BIT  // Channel 48
            output Application.Provision_2.RL1_output_operation_write_int : WORD  // Channel 48.Channel 48
            output Application.Provision_2.set_param_trigger.Q : BIT  // Channel 49
            output Application.Provision_2.RL2_output_operation_write_int : WORD  // Channel 49.Channel 49
            output Application.Provision_2.set_param_trigger.Q : BIT  // Channel 50
            output Application.Provision_2.RL3_output_operation_write_int : WORD  // Channel 50.Channel 50
            output Application.Provision_2.set_param_trigger.Q : BIT  // Channel 51
            output Application.Provision_2.RL4_output_operation_write_int : WORD  // Channel 51.Channel 51
            output Application.Provision_2.Door_stop_timeout_write_int : WORD  // Channel 52.Channel 52
            output Application.Provision_2.set_param_trigger.Q : BIT  // Channel 53
            output Application.Provision_2.DI1_digital_input_operation_write_int : WORD  // Channel 53.Channel 53
            output Application.Provision_2.set_param_trigger.Q : BIT  // Channel 54
            output Application.Provision_2.DI1_digital_input_activation_write_int : WORD  // Channel 54.Channel 54
            output Application.Provision_2.set_param_trigger.Q : BIT  // Channel 55
            output Application.Provision_2.DI2_digital_input_operation_write_int : WORD  // Channel 55.Channel 55
            output Application.Provision_2.set_param_trigger.Q : BIT  // Channel 56
            output Application.Provision_2.DI2_digital_input_activation_write_int : WORD  // Channel 56.Channel 56
            output Application.Provision_2.set_param_trigger.Q : BIT  // Channel 57
            output Application.Provision_2.Light_control_mode_write_int : WORD  // Channel 57.Channel 57
            output Application.Provision_2.set_param_trigger.Q : BIT  // Channel 58
            output Application.Provision_2.Defrost_time_optimization_write_int : WORD  // Channel 58.Channel 58
            unmapped channels: Channel 0, Channel 1, Channel 2, Channel 3, Channel 4, Channel 5, Channel 6, Channel 7, Channel 8, Channel 9, Channel 10, Channel 11, Channel 12, Channel 13, Channel 14, Channel 15, Channel 16, Channel 17, Channel 18, Channel 18, Channel 19, Channel 20, Channel 21, Channel 22, Channel 23, Channel 24, Channel 25, Channel 25, Channel 26, Channel 27, Channel 28, Channel 29, Channel 30, Channel 31, Channel 32, Channel 33, Channel 34, Channel 35, Channel 36, Channel 37,
              Channel 38, Channel 45, Channel 39, Channel 40, Channel 41, Channel 42, Channel 43, Channel 44, Channel 46, Channel 47, Channel 48, Channel 49, Channel 50, Channel 51, Channel 52, Channel 53, Channel 54, Channel 55, Channel 56, Channel 57, Channel 58
        Modbus_Slave_COM_Prov3 : Modbus Server, COM Port, CODESYS, version 4.4.0.0
            settings: SlaveAddress = 3; ResponseTimeout = 1000; UseExtendedFunctionCodes = TRUE; Channel 0.Function Code = 3; Channel 0.Read Offset = 16#0000; Channel 0.Read Length = 18; Channel 0.Write Offset = 0; Channel 0.Write Length = 0; Channel 0.Cycle Time = 100; Channel 1.Function Code = 3; Channel 1.Read Offset = 16#0064; Channel 1.Read Length = 3; Channel 1.Write Offset = 0; Channel 1.Write Length = 0; Channel 1.Cycle Time = 100; Channel 2.Function Code = 3; Channel 2.Read Offset = 16#00C8; Channel 2.Read Length = 11; Channel 2.Write Offset = 0; Channel 2.Write Length = 0; Channel 2.Cycle Time = 100; Channel 3.Function Code = 3; Channel 3.Read Offset = 16#012C; Channel 3.Read Length = 10; Channel 3.Write Offset = 0; Channel 3.Write Length = 0; Channel 3.Cycle Time = 100; Channel 4.Function Code = 3; Channel 4.Read Offset = 16#0190; Channel 4.Read Length = 13; Channel 4.Write Offset = 0; Channel 4.Write Length = 0; Channel 4.Cycle Time = 100; Channel 5.Function Code = 3; Channel 5.Read Offset = 16#01F4; Channel 5.Read Length = 9; Channel 5.Write Offset = 0; Channel 5.Write Length = 0; Channel 5.Cycle Time = 100; Channel 6.Function Code = 3;
              Channel 6.Read Offset = 16#0258; Channel 6.Read Length = 10; Channel 6.Write Offset = 0; Channel 6.Write Length = 0; Channel 6.Cycle Time = 100; Channel 7.Function Code = 3; Channel 7.Read Offset = 16#02BE; Channel 7.Read Length = 2; Channel 7.Write Offset = 0; Channel 7.Write Length = 0; Channel 7.Cycle Time = 100; Channel 8.Function Code = 3; Channel 8.Read Offset = 16#01C2; Channel 8.Read Length = 8; Channel 8.Write Offset = 0; Channel 8.Write Length = 0; Channel 8.Cycle Time = 100; Channel 9.Function Code = 3; Channel 9.Read Offset = 16#00C1; Channel 9.Read Length = 5; Channel 9.Write Offset = 0; Channel 9.Write Length = 0; Channel 9.Cycle Time = 100; Channel 10.Function Code = 3; Channel 10.Read Offset = 16#028A; Channel 10.Read Length = 4; Channel 10.Write Offset = 0; Channel 10.Write Length = 0; Channel 10.Cycle Time = 100; Channel 11.Function Code = 6; Channel 11.Read Offset = 0; Channel 11.Read Length = 0; Channel 11.Write Offset = 16#012F; Channel 11.Write Length = 1; Channel 11.Cycle Time = 100; Channel 12.Function Code = 6; Channel 12.Read Offset = 0; Channel 12.Read Length = 0; Channel 12.Write Offset = 16#02BE; Channel 12.Write Length = 1;
              Channel 12.Cycle Time = 100; Channel 13.Function Code = 6; Channel 13.Read Offset = 0; Channel 13.Read Length = 0; Channel 13.Write Offset = 16#0130; Channel 13.Write Length = 1; Channel 13.Cycle Time = 100; Channel 14.Function Code = 6; Channel 14.Read Offset = 0; Channel 14.Read Length = 0; Channel 14.Write Offset = 16#0131; Channel 14.Write Length = 1; Channel 14.Cycle Time = 100; Channel 15.Function Code = 6; Channel 15.Read Offset = 0; Channel 15.Read Length = 0; Channel 15.Write Offset = 16#01F5; Channel 15.Write Length = 1; Channel 15.Cycle Time = 100; Channel 16.Function Code = 6; Channel 16.Read Offset = 0; Channel 16.Read Length = 0; Channel 16.Write Offset = 16#01F6; Channel 16.Write Length = 1; Channel 16.Cycle Time = 100; Channel 17.Function Code = 6; Channel 17.Read Offset = 0; Channel 17.Read Length = 0; Channel 17.Write Offset = 16#0079; Channel 17.Write Length = 1; Channel 17.Cycle Time = 100; Channel 18.Function Code = 6; Channel 18.Read Offset = 0; Channel 18.Read Length = 0; Channel 18.Write Offset = 16#0080; Channel 18.Write Length = 1; Channel 18.Cycle Time = 100; Channel 19.Function Code = 6; Channel 19.Read Offset = 0; Channel 19.Read Length = 0;
              Channel 19.Write Offset = 16#0191; Channel 19.Write Length = 1; Channel 19.Cycle Time = 100; Channel 20.Function Code = 6; Channel 20.Read Offset = 0; Channel 20.Read Length = 0; Channel 20.Write Offset = 16#0196; Channel 20.Write Length = 1; Channel 20.Cycle Time = 100; Channel 21.Function Code = 6; Channel 21.Read Offset = 0; Channel 21.Read Length = 0; Channel 21.Write Offset = 16#0198; Channel 21.Write Length = 1; Channel 21.Cycle Time = 100; Channel 22.Function Code = 6; Channel 22.Read Offset = 0; Channel 22.Read Length = 0; Channel 22.Write Offset = 16#0197; Channel 22.Write Length = 1; Channel 22.Cycle Time = 100; Channel 23.Function Code = 6; Channel 23.Read Offset = 0; Channel 23.Read Length = 0; Channel 23.Write Offset = 16#007A; Channel 23.Write Length = 1; Channel 23.Cycle Time = 100; Channel 24.Function Code = 6; Channel 24.Read Offset = 0; Channel 24.Read Length = 0; Channel 24.Write Offset = 16#01C2; Channel 24.Write Length = 1; Channel 24.Cycle Time = 100; Channel 25.Function Code = 6; Channel 25.Read Offset = 0; Channel 25.Read Length = 0; Channel 25.Write Offset = 16#00C8; Channel 25.Write Length = 1; Channel 25.Cycle Time = 100; Channel 26.Function Code = 6;
              Channel 26.Read Offset = 0; Channel 26.Read Length = 0; Channel 26.Write Offset = 16#012C; Channel 26.Write Length = 1; Channel 26.Cycle Time = 100; Channel 27.Function Code = 6; Channel 27.Read Offset = 0; Channel 27.Read Length = 0; Channel 27.Write Offset = 16#012D; Channel 27.Write Length = 1; Channel 27.Cycle Time = 100; Channel 28.Function Code = 6; Channel 28.Read Offset = 0; Channel 28.Read Length = 0; Channel 28.Write Offset = 16#012E; Channel 28.Write Length = 1; Channel 28.Cycle Time = 100; Channel 29.Function Code = 6; Channel 29.Read Offset = 0; Channel 29.Read Length = 0; Channel 29.Write Offset = 16#0132; Channel 29.Write Length = 1; Channel 29.Cycle Time = 100; Channel 30.Function Code = 6; Channel 30.Read Offset = 0; Channel 30.Read Length = 0; Channel 30.Write Offset = 16#0133; Channel 30.Write Length = 1; Channel 30.Cycle Time = 100; Channel 31.Function Code = 6; Channel 31.Read Offset = 0; Channel 31.Read Length = 0; Channel 31.Write Offset = 16#0134; Channel 31.Write Length = 1; Channel 31.Cycle Time = 100; Channel 32.Function Code = 6; Channel 32.Read Offset = 0; Channel 32.Read Length = 0; Channel 32.Write Offset = 16#0135; Channel 32.Write Length = 1;
              Channel 32.Cycle Time = 100; Channel 33.Function Code = 6; Channel 33.Read Offset = 0; Channel 33.Read Length = 0; Channel 33.Write Offset = 16#0192; Channel 33.Write Length = 1; Channel 33.Cycle Time = 100; Channel 34.Function Code = 6; Channel 34.Read Offset = 0; Channel 34.Read Length = 0; Channel 34.Write Offset = 16#0194; Channel 34.Write Length = 1; Channel 34.Cycle Time = 100; Channel 35.Function Code = 6; Channel 35.Read Offset = 0; Channel 35.Read Length = 0; Channel 35.Write Offset = 16#019C; Channel 35.Write Length = 1; Channel 35.Cycle Time = 100; Channel 36.Function Code = 6; Channel 36.Read Offset = 0; Channel 36.Read Length = 0; Channel 36.Write Offset = 16#019A; Channel 36.Write Length = 1; Channel 36.Cycle Time = 100; Channel 37.Function Code = 6; Channel 37.Read Offset = 0; Channel 37.Read Length = 0; Channel 37.Write Offset = 16#019B; Channel 37.Write Length = 1; Channel 37.Cycle Time = 100; Channel 45.Function Code = 6; Channel 45.Read Offset = 0; Channel 45.Read Length = 0; Channel 45.Write Offset = 16#01F4; Channel 45.Write Length = 1; Channel 45.Cycle Time = 100; Channel 39.Function Code = 6; Channel 39.Read Offset = 0; Channel 39.Read Length = 0;
              Channel 39.Write Offset = 16#01C3; Channel 39.Write Length = 1; Channel 39.Cycle Time = 100; Channel 40.Function Code = 6; Channel 40.Read Offset = 0; Channel 40.Read Length = 0; Channel 40.Write Offset = 16#01C4; Channel 40.Write Length = 1; Channel 40.Cycle Time = 100; Channel 41.Function Code = 6; Channel 41.Read Offset = 0; Channel 41.Read Length = 0; Channel 41.Write Offset = 16#01FA; Channel 41.Write Length = 1; Channel 41.Cycle Time = 100; Channel 42.Function Code = 6; Channel 42.Read Offset = 0; Channel 42.Read Length = 0; Channel 42.Write Offset = 16#0259; Channel 42.Write Length = 1; Channel 42.Cycle Time = 100; Channel 43.Function Code = 6; Channel 43.Read Offset = 0; Channel 43.Read Length = 0; Channel 43.Write Offset = 16#025A; Channel 43.Write Length = 1; Channel 43.Cycle Time = 100; Channel 44.Function Code = 6; Channel 44.Read Offset = 0; Channel 44.Read Length = 0; Channel 44.Write Offset = 16#025B; Channel 44.Write Length = 1; Channel 44.Cycle Time = 100; Channel 46.Function Code = 6; Channel 46.Read Offset = 0; Channel 46.Read Length = 0; Channel 46.Write Offset = 16#01F4; Channel 46.Write Length = 1; Channel 46.Cycle Time = 100; Channel 47.Function Code = 6;
              Channel 47.Read Offset = 0; Channel 47.Read Length = 0; Channel 47.Write Offset = 16#00D0; Channel 47.Write Length = 1; Channel 47.Cycle Time = 100; Channel 48.Function Code = 6; Channel 48.Read Offset = 0; Channel 48.Read Length = 0; Channel 48.Write Offset = 16#028A; Channel 48.Write Length = 1; Channel 48.Cycle Time = 100; Channel 49.Function Code = 6; Channel 49.Read Offset = 0; Channel 49.Read Length = 0; Channel 49.Write Offset = 16#028B; Channel 49.Write Length = 1; Channel 49.Cycle Time = 100; Channel 50.Function Code = 6; Channel 50.Read Offset = 0; Channel 50.Read Length = 0; Channel 50.Write Offset = 16#028C; Channel 50.Write Length = 1; Channel 50.Cycle Time = 100; Channel 51.Function Code = 6; Channel 51.Read Offset = 0; Channel 51.Read Length = 0; Channel 51.Write Offset = 16#028D; Channel 51.Write Length = 1; Channel 51.Cycle Time = 100; Channel 52.Function Code = 6; Channel 52.Read Offset = 0; Channel 52.Read Length = 0; Channel 52.Write Offset = 16#025C; Channel 52.Write Length = 1; Channel 52.Cycle Time = 100; Channel 53.Function Code = 6; Channel 53.Read Offset = 0; Channel 53.Read Length = 0; Channel 53.Write Offset = 16#025D; Channel 53.Write Length = 1;
              Channel 53.Cycle Time = 100; Channel 54.Function Code = 6; Channel 54.Read Offset = 0; Channel 54.Read Length = 0; Channel 54.Write Offset = 16#025E; Channel 54.Write Length = 1; Channel 54.Cycle Time = 100; Channel 55.Function Code = 6; Channel 55.Read Offset = 0; Channel 55.Read Length = 0; Channel 55.Write Offset = 16#025F; Channel 55.Write Length = 1; Channel 55.Cycle Time = 100; Channel 56.Function Code = 6; Channel 56.Read Offset = 0; Channel 56.Read Length = 0; Channel 56.Write Offset = 16#0260; Channel 56.Write Length = 1; Channel 56.Cycle Time = 100; Channel 57.Function Code = 6; Channel 57.Read Offset = 0; Channel 57.Read Length = 0; Channel 57.Write Offset = 16#0261; Channel 57.Write Length = 1; Channel 57.Cycle Time = 100; Channel 58.Function Code = 6; Channel 58.Read Offset = 0; Channel 58.Read Length = 0; Channel 58.Write Offset = 16#0193; Channel 58.Write Length = 1; Channel 58.Cycle Time = 100
            input  Application.Main_program.modbus_var[3,0] : WORD  // Channel 0.Channel 0
            input  Application.Main_program.modbus_var[3,1] : WORD  // Channel 0.Channel 0
            input  Application.Main_program.modbus_var[3,2] : WORD  // Channel 0.Channel 0
            input  Application.Main_program.modbus_var[3,3] : WORD  // Channel 0.Channel 0
            input  Application.Main_program.modbus_var[3,4] : WORD  // Channel 0.Channel 0
            input  Application.Main_program.modbus_var[3,5] : WORD  // Channel 0.Channel 0
            input  Application.Main_program.modbus_var[3,6] : WORD  // Channel 0.Channel 0
            input  Application.Main_program.modbus_var[3,7] : WORD  // Channel 0.Channel 0
            input  Application.Main_program.modbus_var[3,8] : WORD  // Channel 0.Channel 0
            input  Application.Main_program.modbus_var[3,9] : WORD  // Channel 0.Channel 0
            input  Application.Main_program.modbus_var[3,10] : WORD  // Channel 0.Channel 0
            input  Application.Main_program.modbus_var[3,11] : WORD  // Channel 0.Channel 0
            input  Application.Main_program.modbus_var[3,12] : WORD  // Channel 0.Channel 0
            input  Application.Main_program.modbus_var[3,13] : WORD  // Channel 0.Channel 0
            input  Application.Main_program.modbus_var[3,14] : WORD  // Channel 0.Channel 0
            input  Application.Main_program.modbus_var[3,15] : WORD  // Channel 0.Channel 0
            input  Application.Main_program.modbus_var[3,16] : WORD  // Channel 0.Channel 0
            input  Application.Main_program.modbus_var[3,17] : WORD  // Channel 0.Channel 0
            input  Application.Main_program.modbus_var[3,100] : WORD  // Channel 1.Channel 1
            input  Application.Main_program.modbus_var[3,101] : WORD  // Channel 1.Channel 1
            input  Application.Main_program.modbus_var[3,102] : WORD  // Channel 1.Channel 1
            output Application.Provision_3.get_param_trigger.Q : BIT  // Channel 2
            input  Application.Main_program.modbus_var[3,200] : WORD  // Channel 2.Channel 2
            input  Application.Main_program.modbus_var[3,201] : WORD  // Channel 2.Channel 2
            input  Application.Main_program.modbus_var[3,202] : WORD  // Channel 2.Channel 2
            input  Application.Main_program.modbus_var[3,203] : WORD  // Channel 2.Channel 2
            input  Application.Main_program.modbus_var[3,204] : WORD  // Channel 2.Channel 2
            input  Application.Main_program.modbus_var[3,205] : WORD  // Channel 2.Channel 2
            input  Application.Main_program.modbus_var[3,206] : WORD  // Channel 2.Channel 2
            input  Application.Main_program.modbus_var[3,207] : WORD  // Channel 2.Channel 2
            input  Application.Main_program.modbus_var[3,208] : WORD  // Channel 2.Channel 2
            input  Application.Main_program.modbus_var[3,209] : WORD  // Channel 2.Channel 2
            input  Application.Main_program.modbus_var[3,210] : WORD  // Channel 2.Channel 2
            input  Application.Main_program.modbus_var[3,300] : WORD  // Channel 3.Channel 3
            input  Application.Main_program.modbus_var[3,301] : WORD  // Channel 3.Channel 3
            input  Application.Main_program.modbus_var[3,302] : WORD  // Channel 3.Channel 3
            input  Application.Main_program.modbus_var[3,303] : WORD  // Channel 3.Channel 3
            input  Application.Main_program.modbus_var[3,304] : WORD  // Channel 3.Channel 3
            input  Application.Main_program.modbus_var[3,305] : WORD  // Channel 3.Channel 3
            input  Application.Main_program.modbus_var[3,306] : WORD  // Channel 3.Channel 3
            input  Application.Main_program.modbus_var[3,307] : WORD  // Channel 3.Channel 3
            input  Application.Main_program.modbus_var[3,308] : WORD  // Channel 3.Channel 3
            input  Application.Main_program.modbus_var[3,309] : WORD  // Channel 3.Channel 3
            input  Application.Main_program.modbus_var[3,400] : WORD  // Channel 4.Channel 4
            input  Application.Main_program.modbus_var[3,401] : WORD  // Channel 4.Channel 4
            input  Application.Main_program.modbus_var[3,402] : WORD  // Channel 4.Channel 4
            input  Application.Main_program.modbus_var[3,403] : WORD  // Channel 4.Channel 4
            input  Application.Main_program.modbus_var[3,404] : WORD  // Channel 4.Channel 4
            input  Application.Main_program.modbus_var[3,405] : WORD  // Channel 4.Channel 4
            input  Application.Main_program.modbus_var[3,406] : WORD  // Channel 4.Channel 4
            input  Application.Main_program.modbus_var[3,407] : WORD  // Channel 4.Channel 4
            input  Application.Main_program.modbus_var[3,408] : WORD  // Channel 4.Channel 4
            input  Application.Main_program.modbus_var[3,409] : WORD  // Channel 4.Channel 4
            input  Application.Main_program.modbus_var[3,410] : WORD  // Channel 4.Channel 4
            input  Application.Main_program.modbus_var[3,411] : WORD  // Channel 4.Channel 4
            input  Application.Main_program.modbus_var[3,412] : WORD  // Channel 4.Channel 4
            input  Application.Main_program.modbus_var[3,500] : WORD  // Channel 5.Channel 5
            input  Application.Main_program.modbus_var[3,501] : WORD  // Channel 5.Channel 5
            input  Application.Main_program.modbus_var[3,502] : WORD  // Channel 5.Channel 5
            input  Application.Main_program.modbus_var[3,503] : WORD  // Channel 5.Channel 5
            input  Application.Main_program.modbus_var[3,504] : WORD  // Channel 5.Channel 5
            input  Application.Main_program.modbus_var[3,505] : WORD  // Channel 5.Channel 5
            input  Application.Main_program.modbus_var[3,506] : WORD  // Channel 5.Channel 5
            input  Application.Main_program.modbus_var[3,507] : WORD  // Channel 5.Channel 5
            input  Application.Main_program.modbus_var[3,508] : WORD  // Channel 5.Channel 5
            output Application.Provision_3.get_param_trigger.Q : BIT  // Channel 6
            input  Application.Main_program.modbus_var[3,600] : WORD  // Channel 6.Channel 6
            input  Application.Main_program.modbus_var[3,601] : WORD  // Channel 6.Channel 6
            input  Application.Main_program.modbus_var[3,602] : WORD  // Channel 6.Channel 6
            input  Application.Main_program.modbus_var[3,603] : WORD  // Channel 6.Channel 6
            input  Application.Main_program.modbus_var[3,604] : WORD  // Channel 6.Channel 6
            input  Application.Main_program.modbus_var[3,605] : WORD  // Channel 6.Channel 6
            input  Application.Main_program.modbus_var[3,606] : WORD  // Channel 6.Channel 6
            input  Application.Main_program.modbus_var[3,607] : WORD  // Channel 6.Channel 6
            input  Application.Main_program.modbus_var[3,608] : WORD  // Channel 6.Channel 6
            input  Application.Main_program.modbus_var[3,609] : WORD  // Channel 6.Channel 6
            output Application.Provision_3.get_param_trigger.Q : BIT  // Channel 7
            input  Application.Main_program.modbus_var[3,702] : WORD  // Channel 7.Channel 7
            input  Application.Main_program.modbus_var[3,703] : WORD  // Channel 7.Channel 7
            output Application.Provision_3.get_param_trigger.Q : BIT  // Channel 8
            input  Application.Main_program.modbus_var[3,450] : WORD  // Channel 8.Channel 8
            input  Application.Main_program.modbus_var[3,451] : WORD  // Channel 8.Channel 8
            input  Application.Main_program.modbus_var[3,452] : WORD  // Channel 8.Channel 8
            input  Application.Main_program.modbus_var[3,453] : WORD  // Channel 8.Channel 8
            input  Application.Main_program.modbus_var[3,454] : WORD  // Channel 8.Channel 8
            input  Application.Main_program.modbus_var[3,455] : WORD  // Channel 8.Channel 8
            input  Application.Main_program.modbus_var[3,456] : WORD  // Channel 8.Channel 8
            input  Application.Main_program.modbus_var[3,457] : WORD  // Channel 8.Channel 8
            output Application.Provision_3.get_param_trigger.Q : BIT  // Channel 9
            output Application.Provision_3.get_param_trigger.Q : BIT  // Channel 10
            input  Application.Main_program.modbus_var[3,650] : WORD  // Channel 10.Channel 10
            input  Application.Main_program.modbus_var[3,651] : WORD  // Channel 10.Channel 10
            input  Application.Main_program.modbus_var[3,652] : WORD  // Channel 10.Channel 10
            input  Application.Main_program.modbus_var[3,653] : WORD  // Channel 10.Channel 10
            output Application.Provision_3.write_data_setp.Q : BIT  // Channel 11
            output Application.Provision_3.setp_write_word : WORD  // Channel 11.Channel 11
            output Application.Provision_3.write_data_control.Q : BIT  // Channel 12
            output Application.Provision_3.standby_write : WORD  // Channel 12.Channel 12
            output Application.Provision_3.write_data_setp.Q : BIT  // Channel 13
            output Application.Provision_3.Thermostat_OFF_ON_write_word : WORD  // Channel 13.Channel 13
            output Application.Provision_3.write_data_setp.Q : BIT  // Channel 14
            output Application.Provision_3.Thermostat_ON_OFF_write_word : WORD  // Channel 14.Channel 14
            output Application.Provision_3.write_data_alarm.Q : BIT  // Channel 15
            output Application.Provision_3.Low_temperature_alarm_thres_write_word : WORD  // Channel 15.Channel 15
            output Application.Provision_3.write_data_alarm.Q : BIT  // Channel 16
            output Application.Provision_3.High_temperature_alarm_thres_write_word : WORD  // Channel 16.Channel 16
            output Application.Provision_3.write_data_mute.Q : BIT  // Channel 17
            output Application.Provision_3.muteAlarm : WORD  // Channel 17.Channel 17
            output Application.Provision_3.Time_based_defrost_write_word : WORD  // Channel 18.Channel 18
            output Application.Provision_3.write_data_defrost.Q : BIT  // Channel 19
            output Application.Provision_3.Time_based_defrost_write_word : WORD  // Channel 19.Channel 19
            output Application.Provision_3.write_data_defrost.Q : BIT  // Channel 20
            output Application.Provision_3.Defrost_end_temperature_write_word : WORD  // Channel 20.Channel 20
            output Application.Provision_3.write_data_defrost.Q : BIT  // Channel 21
            output Application.Provision_3.Drain_down_time_write_int : WORD  // Channel 21.Channel 21
            output Application.Provision_3.write_data_defrost.Q : BIT  // Channel 22
            output Application.Provision_3.Maximum_defrost_duration_write_word : WORD  // Channel 22.Channel 22
            output Application.Provision_3.write_data_man_defrost.Q : BIT  // Channel 23
            output Application.Provision_3.defrost_write : WORD  // Channel 23.Channel 23
            output Application.Provision_3.set_param_trigger.Q : BIT  // Channel 24
            output Application.Provision_3.Fan_stop_temperature_write_word : WORD  // Channel 24.Channel 24
            output Application.Provision_3.preset_parameters_write_int : WORD  // Channel 25.Channel 25
            output Application.Provision_3.set_param_trigger.Q : BIT  // Channel 26
            output Application.Provision_3.Readout_scale_write_int : WORD  // Channel 26.Channel 26
            output Application.Provision_3.set_param_trigger.Q : BIT  // Channel 27
            output Application.Provision_3.Minimum_temperature_setpoint_write_int : WORD  // Channel 27.Channel 27
            output Application.Provision_3.set_param_trigger.Q : BIT  // Channel 28
            output Application.Provision_3.Maximum_temperature_setpoint_write_int : WORD  // Channel 28.Channel 28
            output Application.Provision_3.set_param_trigger.Q : BIT  // Channel 29
            output Application.Provision_3.CH_minimum_OFF_time_write_int : WORD  // Channel 29.Channel 29
            output Application.Provision_3.set_param_trigger.Q : BIT  // Channel 30
            output Application.Provision_3.CH_minimum_ON_time_write_int : WORD  // Channel 30.Channel 30
            output Application.Provision_3.set_param_trigger.Q : BIT  // Channel 31
            output Application.Provision_3.CH_output_ON_when_probe_T1_is_faulty_write_int : WORD  // Channel 31.Channel 31
            output Application.Provision_3.set_param_trigger.Q : BIT  // Channel 32
            output Application.Provision_3.CH_output_OFF_when_probe_T1_is_faulty_write_int : WORD  // Channel 32.Channel 32
            output Application.Provision_3.set_param_trigger.Q : BIT  // Channel 33
            output Application.Provision_3.Minimum_Time_Between_Defrost_write_int : WORD  // Channel 33.Channel 33
            output Application.Provision_3.set_param_trigger.Q : BIT  // Channel 34
            output Application.Provision_3.Defrost_type_write_int : WORD  // Channel 34.Channel 34
            output Application.Provision_3.set_param_trigger.Q : BIT  // Channel 35
            output Application.Provision_3.Fan_restart_temperature_after_defrost_write_int : WORD  // Channel 35.Channel 35
            output Application.Provision_3.set_param_trigger.Q : BIT  // Channel 36
            output Application.Provision_3.Display_delay_write_int : WORD  // Channel 36.Channel 36
            output Application.Provision_3.set_param_trigger.Q : BIT  // Channel 37
            output Application.Provision_3.Fans_active_during_defrost_write_int : WORD  // Channel 37.Channel 37
            output Application.Provision_3.set_param_trigger.Q : BIT  // Channel 39
            output Application.Provision_3.Maximum_fan_stop_for_FDD_FET_write_int : WORD  // Channel 39.Channel 39
            output Application.Provision_3.set_param_trigger.Q : BIT  // Channel 40
            output Application.Provision_3.Fan_mode_during_thermostatic_control_write_int : WORD  // Channel 40.Channel 40
            output Application.Provision_3.set_param_trigger.Q : BIT  // Channel 41
            output Application.Provision_3.Temperature_alarm_delay_write_int : WORD  // Channel 41.Channel 41
            output Application.Provision_3.set_param_trigger.Q : BIT  // Channel 42
            output Application.Provision_3.Door_switch_input_mode_write_int : WORD  // Channel 42.Channel 42
            output Application.Provision_3.set_param_trigger.Q : BIT  // Channel 43
            output Application.Provision_3.Door_alarm_delay_write_int : WORD  // Channel 43.Channel 43
            output Application.Provision_3.set_param_trigger.Q : BIT  // Channel 44
            output Application.Provision_3.Compressor_stop_delay_write_int : WORD  // Channel 44.Channel 44
            output Application.Provision_3.set_param_trigger.Q : BIT  // Channel 46
            output Application.Provision_3.Alarm_threshold_management_write_int : WORD  // Channel 46.Channel 46
            output Application.Provision_3.set_param_trigger.Q : BIT  // Channel 47
            output Application.Provision_3.Display_slowdown_write_int : WORD  // Channel 47.Channel 47
            output Application.Provision_3.set_param_trigger.Q : BIT  // Channel 48
            output Application.Provision_3.RL1_output_operation_write_int : WORD  // Channel 48.Channel 48
            output Application.Provision_3.set_param_trigger.Q : BIT  // Channel 49
            output Application.Provision_3.RL2_output_operation_write_int : WORD  // Channel 49.Channel 49
            output Application.Provision_3.set_param_trigger.Q : BIT  // Channel 50
            output Application.Provision_3.RL3_output_operation_write_int : WORD  // Channel 50.Channel 50
            output Application.Provision_3.set_param_trigger.Q : BIT  // Channel 51
            output Application.Provision_3.RL4_output_operation_write_int : WORD  // Channel 51.Channel 51
            output Application.Provision_3.Door_stop_timeout_write_int : WORD  // Channel 52.Channel 52
            output Application.Provision_3.set_param_trigger.Q : BIT  // Channel 53
            output Application.Provision_3.DI1_digital_input_operation_write_int : WORD  // Channel 53.Channel 53
            output Application.Provision_3.set_param_trigger.Q : BIT  // Channel 54
            output Application.Provision_3.DI1_digital_input_activation_write_int : WORD  // Channel 54.Channel 54
            output Application.Provision_3.set_param_trigger.Q : BIT  // Channel 55
            output Application.Provision_3.DI2_digital_input_operation_write_int : WORD  // Channel 55.Channel 55
            output Application.Provision_3.set_param_trigger.Q : BIT  // Channel 56
            output Application.Provision_3.DI2_digital_input_activation_write_int : WORD  // Channel 56.Channel 56
            output Application.Provision_3.set_param_trigger.Q : BIT  // Channel 57
            output Application.Provision_3.Light_control_mode_write_int : WORD  // Channel 57.Channel 57
            output Application.Provision_3.set_param_trigger.Q : BIT  // Channel 58
            output Application.Provision_3.Defrost_time_optimization_write_int : WORD  // Channel 58.Channel 58
            unmapped channels: Channel 0, Channel 1, Channel 2, Channel 3, Channel 4, Channel 5, Channel 6, Channel 7, Channel 8, Channel 9, Channel 10, Channel 11, Channel 12, Channel 13, Channel 14, Channel 15, Channel 16, Channel 17, Channel 18, Channel 18, Channel 19, Channel 20, Channel 21, Channel 22, Channel 23, Channel 24, Channel 25, Channel 25, Channel 26, Channel 27, Channel 28, Channel 29, Channel 30, Channel 31, Channel 32, Channel 33, Channel 34, Channel 35, Channel 36, Channel 37,
              Channel 38, Channel 45, Channel 39, Channel 40, Channel 41, Channel 42, Channel 43, Channel 44, Channel 46, Channel 47, Channel 48, Channel 49, Channel 50, Channel 51, Channel 52, Channel 53, Channel 54, Channel 55, Channel 56, Channel 57, Channel 58
    SoftMotion General Axis Pool
  AC_GENERATOR_DATA
  text list GlobalTextList
*)

// Device/Application/Main_program
PROGRAM Main_program
VAR CONSTANT
	c_iNUM_ROOM : INT := 2;
END_VAR
VAR
	modbus_var : ARRAY[0..100,0..800] OF WORD;
	Provision_room1 : FB_Provision_room;
	Provision_room2 : FB_Provision_room;
	Provision_room3 : FB_Provision_room;
	Prov1 : clsLampFunction;
	Prov2 : clsLampFunction;
	status_switch : BOOL;
	text_message : STRING;
	test1 : WORD ;
	test2 : WORD ;
	test3 : WORD ;
	test4 : WORD ;

END_VAR

(* Initialize all of the rooms *)
Prov1(prov_name :='Provision1');
Prov2(prov_name :='Provision2');
text_message:= 'testmessage';

test1 := modbus_var[1,0] ;
test2 := modbus_var[1,1] ;
test3 := modbus_var[2,0] ;
test4 := modbus_var[2,1] ;

Provision_room1(I_Provision_name:='1-Wine & Beer',I_Modbus_var := modbus_var,I_Provision_Room := 1);
Provision_room2(I_Provision_name:='2 - Red Wine',I_Modbus_var := modbus_var,I_Provision_Room := 2);
Provision_room3(I_Provision_name:='3 - Cooked Food',I_Modbus_var := modbus_var,I_Provision_Room := 3);

END_PROGRAM

// Device/Application/FB_Provision_room
FUNCTION_BLOCK FB_Provision_room IMPLEMENTS ITF_provision_room
VAR_INPUT
	I_modbus_var : ARRAY[0..100,0..800] OF WORD;
	I_Provision_Room : INT;
	I_Provision_name : STRING ;
	I_alarm : BOOL;
	I_Machine_standby : BOOL;
	I_Room_temp : REAL ;
	I_Setpoint : REAL ;
END_VAR

VAR_OUTPUT
	O_write_data_setp : R_TRIG;
	O_word_setpoint : WORD;
END_VAR
VAR
	xTrigger_setpoint : BOOL ;
	setpoint_write : REAL ;
END_VAR

METHOD MET_assign_values : BOOL
VAR_OUTPUT

END_VAR
END_METHOD

{warning 'Add property implementation'}
PROPERTY P_Alarm : BOOL
GET
P_Alarm := maskbitFunction(I_modbus_var[I_provision_room,100],0);
END_GET
SET
END_SET
END_PROPERTY

PROPERTY P_Defrost : bool
GET
P_Defrost:= maskbitFunction(I_modbus_var[I_provision_room,100],2);
END_GET
SET
END_SET
END_PROPERTY

PROPERTY P_Defrost_end_temperature : real
GET
P_Defrost_end_temperature:=scaleFunction(I_modbus_var[I_provision_room,406],0.1, 0);
END_GET
SET
END_SET
END_PROPERTY

PROPERTY P_Door_open : bool
GET
P_Door_open:= maskbitFunction(I_modbus_var[I_provision_room,100],3);
END_GET
SET
END_SET
END_PROPERTY

PROPERTY P_Dout2 : bool
GET
P_Dout2:= maskbitFunction(I_modbus_var[I_provision_room,102],1);
END_GET
SET
END_SET
END_PROPERTY

PROPERTY P_Dout3 : bool
GET
P_Dout3:= maskbitFunction(I_modbus_var[I_provision_room,102],2);
END_GET
SET
END_SET
END_PROPERTY

PROPERTY P_Drain_down_time : real
GET
P_Drain_down_time:= scaleFunction(I_modbus_var[I_provision_room,408],1, 0);
END_GET
SET
END_SET
END_PROPERTY

PROPERTY P_Generic_alarm : bool
GET
P_Generic_alarm:= maskbitFunction(I_modbus_var[I_provision_room,101],6);
END_GET
SET
END_SET
END_PROPERTY

PROPERTY P_High_temperature_alarm_threshold : REAL
GET
P_High_temperature_alarm_threshold := scaleFunction(I_modbus_var[I_provision_room,502],0.1, 0);
END_GET
SET
END_SET
END_PROPERTY

PROPERTY P_High_temperature : bool
GET
P_High_temperature:= maskbitFunction(I_modbus_var[I_provision_room,101],4);
END_GET
SET
END_SET
END_PROPERTY

PROPERTY P_Low_temperature : bool
GET
P_Low_temperature:= maskbitFunction(I_modbus_var[I_provision_room,101],3);
END_GET
SET
END_SET
END_PROPERTY

PROPERTY P_Low_temperature_alarm_threshold : REAL
GET
P_Low_temperature_alarm_threshold := scaleFunction(I_modbus_var[I_provision_room,501],0.1, 0);
END_GET
SET
END_SET
END_PROPERTY

{warning 'Add property implementation'}
PROPERTY P_Machine_standby : BOOL
GET
P_Machine_standby := NOT(maskbitFunction(I_modbus_var[I_provision_room,100],5));
END_GET
SET
END_SET
END_PROPERTY

PROPERTY P_Maximum_defrost_duration : real
GET
P_Maximum_defrost_duration:=scaleFunction(I_modbus_var[I_provision_room,407],1, 0);
END_GET
SET
END_SET
END_PROPERTY

PROPERTY P_Provision_name : STRING
GET
P_Provision_name := I_Provision_name;
END_GET
SET
END_SET
END_PROPERTY

PROPERTY P_Room_temp : REAL
GET
P_Room_temp:= scaleFunction(I_modbus_var[I_provision_room,0],0.1, 0);
END_GET
SET
END_SET
END_PROPERTY

{warning 'Add property implementation'}
PROPERTY P_Setpoint : REAL
GET
P_Setpoint:= scaleFunction(I_modbus_var[I_provision_room,303],0.1, 0);
END_GET
SET
END_SET
END_PROPERTY

PROPERTY P_T1_failure : bool
GET
P_T1_failure := maskbitFunction(I_modbus_var[I_provision_room,101],0);
END_GET
SET
END_SET
END_PROPERTY

PROPERTY P_T2_failure : bool
GET
P_T2_failure := maskbitFunction(I_modbus_var[I_provision_room,101],1);
END_GET
SET
END_SET
END_PROPERTY

PROPERTY P_Temp_defrost : REAL
GET
P_temp_defrost := scaleFunction(I_modbus_var[I_provision_room,0],0.1, 0);
END_GET
SET
END_SET
END_PROPERTY

PROPERTY P_Thermostat_OFF_ON_ref_to_SP : REAL
GET
P_Thermostat_OFF_ON_ref_to_SP := scaleFunction(I_modbus_var[I_provision_room,304],0.1, 0);
END_GET
SET
END_SET
END_PROPERTY

PROPERTY P_Thermostat_ON_OFF_ref_to_SP : REAL
GET
P_Thermostat_ON_OFF_ref_to_SP := scaleFunction(I_modbus_var[I_provision_room,305],1, 0);
END_GET
SET
END_SET
END_PROPERTY

PROPERTY P_Time_based_defrost : real
GET
P_Time_based_defrost:= scaleFunction(I_modbus_var[I_provision_room,401],1, 0);
END_GET
SET
END_SET
END_PROPERTY

METHOD MET_write_sepoint : BOOL
VAR_INPUT
		
END_VAR
VAR
	trigger : BOOL := TRUE ;
	delay_timer : TON ;
END_VAR
O_word_setpoint:= REAL_TO_INT(P_setpoint_write*10) ;
O_write_data_setp(clk:=xTrigger_setpoint);
END_METHOD

PROPERTY P_setpoint_write : REAL ;
GET
VAR
	variable_word : WORD;
END_VAR
P_setpoint_write := setpoint_write ;
END_GET
SET
setpoint_write := P_setpoint_write ;
END_SET
END_PROPERTY

PROPERTY P_test_input : real
GET
P_test_input := P_setpoint_write ;
END_GET
SET
END_SET
END_PROPERTY

PROPERTY P_Thermostat_OFF_ON_ref_to_SP_write : real
GET
END_GET
SET
END_SET
END_PROPERTY

PROPERTY P_Thermostat_ON_OFF_ref_to_SP_write : real
GET
END_GET
SET
END_SET
END_PROPERTY

PROPERTY P_xTrigger_setpoint : bool
GET
VAR
	check_trigger : BOOL := FALSE;
END_VAR
P_xTrigger_setpoint := xTrigger_setpoint;
END_GET
SET
xTrigger_setpoint := P_xTrigger_setpoint ;
MET_write_sepoint();
END_SET
END_PROPERTY

END_FUNCTION_BLOCK

// Device/Application/ITF_provision_room
INTERFACE ITF_provision_room

METHOD MET_assign_values : bool
VAR_OUTPUT
END_VAR
END_METHOD

PROPERTY P_Alarm : bool
GET
END_GET
SET
END_SET
END_PROPERTY

PROPERTY P_Defrost : bool
GET
END_GET
SET
END_SET
END_PROPERTY

PROPERTY P_Defrost_end_temperature : real
GET
END_GET
SET
END_SET
END_PROPERTY

PROPERTY P_Door_open : bool
GET
END_GET
SET
END_SET
END_PROPERTY

PROPERTY P_Dout2 : bool
GET
END_GET
SET
END_SET
END_PROPERTY

PROPERTY P_Dout3 : bool
GET
END_GET
SET
END_SET
END_PROPERTY

PROPERTY P_Drain_down_time : real
GET
END_GET
SET
END_SET
END_PROPERTY

PROPERTY P_Generic_alarm : bool
GET
END_GET
SET
END_SET
END_PROPERTY

PROPERTY P_High_temperature : bool
GET
END_GET
SET
END_SET
END_PROPERTY

PROPERTY P_High_temperature_alarm_threshold : real
GET
END_GET
SET
END_SET
END_PROPERTY

PROPERTY P_Low_temperature : bool
GET
END_GET
SET
END_SET
END_PROPERTY

PROPERTY P_Low_temperature_alarm_threshold : real
GET
END_GET
SET
END_SET
END_PROPERTY

PROPERTY P_Machine_standby : bool
GET
END_GET
SET
END_SET
END_PROPERTY

PROPERTY P_Maximum_defrost_duration : real
GET
END_GET
SET
END_SET
END_PROPERTY

PROPERTY P_Provision_name : string
GET
END_GET
SET
END_SET
END_PROPERTY

PROPERTY P_Room_temp : real
GET
END_GET
SET
END_SET
END_PROPERTY

PROPERTY P_Setpoint : real
GET
END_GET
SET
END_SET
END_PROPERTY

PROPERTY P_T1_failure : bool
GET
END_GET
SET
END_SET
END_PROPERTY

PROPERTY P_T2_failure : bool
GET
END_GET
SET
END_SET
END_PROPERTY

PROPERTY P_Temp_defrost : REAL
GET
END_GET
SET
END_SET
END_PROPERTY

PROPERTY P_Thermostat_OFF_ON_ref_to_SP : real
GET
END_GET
SET
END_SET
END_PROPERTY

PROPERTY P_Thermostat_ON_OFF_ref_to_SP : real
GET
END_GET
SET
END_SET
END_PROPERTY

PROPERTY P_Time_based_defrost : real
GET
END_GET
SET
END_SET
END_PROPERTY

METHOD MET_write_sepoint : Bool
VAR_INPUT
END_VAR
END_METHOD

PROPERTY P_setpoint_write : real
GET
END_GET
SET
END_SET
END_PROPERTY

PROPERTY P_test_input : Real
GET
END_GET
SET
END_SET
END_PROPERTY

PROPERTY P_Thermostat_OFF_ON_ref_to_SP_write : real
GET
END_GET
SET
END_SET
END_PROPERTY

PROPERTY P_Thermostat_ON_OFF_ref_to_SP_write : real
GET
END_GET
SET
END_SET
END_PROPERTY

END_INTERFACE

// Device/Application/Chiller_funct/maskbitFunction
FUNCTION maskbitFunction : BOOL
VAR_INPUT
	inword :WORD;
	bit_no : BYTE;
END_VAR
VAR
END_VAR

maskbitFunction:= EXTRACT(inword, bit_no);

END_FUNCTION

// Device/Application/Chiller_funct/scaleFunction
FUNCTION scaleFunction : REAL
VAR_INPUT
	inValue :INT;
	scaleValue : REAL;
	offsetValue : REAL;
	
END_VAR
VAR_OUTPUT

END_VAR
VAR
	
END_VAR

scaleFunction:=inValue*scaleValue + offsetValue;

END_FUNCTION

// Device/Application/clsLampFunction
FUNCTION_BLOCK clsLampFunction IMPLEMENTS IProvroom
VAR_INPUT
	xLamp : BOOL;
	xSwitch : BOOL;
	prov_name : STRING;
END_VAR
VAR_OUTPUT
	itfProvroom : IProvroom;
END_VAR
VAR
END_VAR


 xLamp:=TRUE;
 //itfLamp.Lamp:=xLamp;

PROPERTY Lamp : BOOL
GET
IF Switch THEN
	Lamp := TRUE;
ELSE 
	Lamp := FALSE;
END_IF;
END_GET
SET
VAR
	xLampOn : BOOL;
END_VAR
 // xLampOn := TRUE;
 // Lamp:=xLampOn;
END_SET
END_PROPERTY

PROPERTY Switch : bool
GET
IF xSwitch THEN
	Switch:= TRUE;
END_IF
END_GET
SET
END_SET
END_PROPERTY

PROPERTY Value : STRING
GET
IF Switch THEN
	Value := prov_name;
ELSE 
	Value := 'False';
END_IF;
END_GET
SET
END_SET
END_PROPERTY

END_FUNCTION_BLOCK

// Device/Application/IProvroom
INTERFACE IProvroom

PROPERTY Lamp : BOOL
GET
END_GET
SET
END_SET
END_PROPERTY

PROPERTY Switch : bool
GET
END_GET
SET
END_SET
END_PROPERTY

PROPERTY Value : string
GET
END_GET
SET
END_SET
END_PROPERTY

END_INTERFACE

// Device/Application/Provision_1
PROGRAM Provision_1
VAR



modbus_var : ARRAY[0..800] OF WORD;
modbus_var1 : ARRAY[2000..2010] OF WORD;
timer_door_open : TON ;
timer_door_closed : TON ;
delay_timer : TON ;
open_time : TIME ;
total_time : TIME ;
opentime_tot : TIME ;
opentime_proc : REAL ;
closetime_tot : TIME ; 
{attribute 'ac_persist' := 'PersistenceChannel'}
set_delaytime : TIME := T#1S;
timer_enable : BOOL;
timer2_enable : BOOL;
timer_elapsed : BOOL ;
start_timer : BOOL := TRUE;
doorclose : F_TRIG;
resettimer_button :BOOL ;
totaltime_ms : LREAL ;
opentime_ms : LREAL ;

temp_provision_room : REAL;
temp_defrost : REAL;
regulator_temp : REAL;

set_point: REAL;
reg2 : REAL ;
reg3 : REAL ;
reg4 : REAL ;
reg5 : REAL ;
reg6 : REAL ;
reg7 : REAL ;
reg8 : REAL ;
reg9 : REAL ;
reg10 : WORD ;
reg11 : REAL ;
reg12 : REAL ;
reg13 : REAL ;
reg14 : REAL ;
reg15 : REAL ;
reg16 : REAL ;
reg17 : REAL ;
T1_offset : REAL ;
T2_offset : REAL ;
T3_offset : REAL ;
T1_span : REAL ;
T2_span : REAL ;
T3_span : REAL ;
valore_tasto1_V : REAL ;
valore_tasto_UP : REAL ;
valore_tasto_DW : REAL ;
valore_tasto_X : REAL ;
Test_display : REAL ;
Tasto_attualmente_premuto : REAL ;
Password : REAL ;

{attribute 'ac_persist' := 'PersistenceChannel'}
preset_parameters : REAL ;
preset_parameters_write_int :INT;
{attribute 'ac_persist' := 'PersistenceChannel'}
Readout_scale : REAL ;
{attribute 'ac_persist' := 'PersistenceChannel'}
Readout_scale_write_int : INT;
{attribute 'ac_persist' := 'PersistenceChannel'}
Minimum_temperature_setpoint : REAL ;
Minimum_temperature_setpoint_write_int : INT ;
{attribute 'ac_persist' := 'PersistenceChannel'}
Maximum_temperature_setpoint : REAL ;
Maximum_temperature_setpoint_write_int : INT ;
setp_write : REAL ;
{attribute 'ac_persist' := 'PersistenceChannel'}
Setpoint : REAL ;
{attribute 'ac_persist' := 'PersistenceChannel'}
Thermostat_OFF_ON_ref_to_SP : REAL  ;
{attribute 'ac_persist' := 'PersistenceChannel'}
Thermostat_ON_OFF_ref_to_SP : REAL  ;
Thermostat_OFF_ON_write : REAL  := 1.0 ;
Thermostat_ON_OFF_write : REAL  := 1.0 ;
Thermostat_OFF_ON_write_word : WORD ;
Thermostat_ON_OFF_write_word : WORD ;
Time_based_defrost_write : REAL   := 8.0  ;
Time_based_defrost_write_word : WORD  ;
Defrost_end_temperature_write : REAL  := 20.0 ;
Defrost_end_temperature_write_word : WORD ;
Fan_restart_temperature_after_defrost_write : REAL ;
Fan_restart_temperature_after_defrost_write_int : INT ;
Maximum_defrost_duration_write : REAL ;
Maximum_defrost_duration_write_word : WORD ;
defrost_write : WORD :=0 ;
{attribute 'ac_persist' := 'PersistenceChannel'}
CH_minimum_OFF_time : REAL ;
CH_minimum_OFF_time_write_int : INT ;
{attribute 'ac_persist' := 'PersistenceChannel'}
CH_minimum_ON_time : REAL ;
CH_minimum_ON_time_write_int : INT ;
{attribute 'ac_persist' := 'PersistenceChannel'}
CH_output_ON_when_probe_T1_is_faulty : REAL ;
CH_output_ON_when_probe_T1_is_faulty_write_int : INT ;
{attribute 'ac_persist' := 'PersistenceChannel'}
CH_output_OFF_when_probe_T1_is_faulty : REAL ;
CH_output_OFF_when_probe_T1_is_faulty_write_int : INT ;

{attribute 'ac_persist' := 'PersistenceChannel'}
Defrost_start_mode : REAL ;
{attribute 'ac_persist' := 'PersistenceChannel'}
Time_based_defrost : REAL ;
{attribute 'ac_persist' := 'PersistenceChannel'}
Minimum_Time_Between_Defrost : REAL ;
Minimum_Time_Between_Defrost_write_int : INT;
{attribute 'ac_persist' := 'PersistenceChannel'}
Defrost_time_optimization : REAL ;
Defrost_time_optimization_write_int : INT;
{attribute 'ac_persist' := 'PersistenceChannel'}
Defrost_type : REAL ;
Defrost_type_write_int : INT;
{attribute 'ac_persist' := 'PersistenceChannel'}
Delay_for_pressure_equalization_for_hot_gas : REAL ;
{attribute 'ac_persist' := 'PersistenceChannel'}
Defrost_end_temperature : REAL ;
{attribute 'ac_persist' := 'PersistenceChannel'}
Maximum_defrost_duration : REAL ;
{attribute 'ac_persist' := 'PersistenceChannel'}
Drain_down_time : REAL ;
Drain_down_time_write : REAL;
Drain_down_time_write_int : INT;
{attribute 'ac_persist' := 'PersistenceChannel'}
Display_defrost_mode : REAL ;
{attribute 'ac_persist' := 'PersistenceChannel'}
Display_delay : REAL ;
Display_delay_write_int : INT;
{attribute 'ac_persist' := 'PersistenceChannel'}
Fans_active_during_defrost : REAL ;
Fans_active_during_defrost_write_int : INT;
{attribute 'ac_persist' := 'PersistenceChannel'}
Fan_restart_temperature_after_defrost : REAL ;
{attribute 'ac_persist' := 'PersistenceChannel'}
Fan_stop_temperature : REAL ;
Fan_stop_temperature_write_int : INT ;
{attribute 'ac_persist' := 'PersistenceChannel'}
Maximum_fan_stop_for_FDD_FET : REAL ;
Maximum_fan_stop_for_FDD_FET_write_int : INT ;
{attribute 'ac_persist' := 'PersistenceChannel'}
Fan_mode_during_thermostatic_control : REAL ;
Fan_mode_during_thermostatic_control_write_int : INT ;
{attribute 'ac_persist' := 'PersistenceChannel'}
Target_evaporator_temperature : REAL ;
{attribute 'ac_persist' := 'PersistenceChannel'}
Fan_stop_delay_after_compressor_stop : REAL ;
{attribute 'ac_persist' := 'PersistenceChannel'}
Timed_fan_stop : REAL ;
{attribute 'ac_persist' := 'PersistenceChannel'}
Timed_fan_run : REAL ;
{attribute 'ac_persist' := 'PersistenceChannel'}
Fan_Minimum_Stop : REAL ;
{attribute 'ac_persist' := 'PersistenceChannel'}
Alarm_threshold_management : REAL ;
Alarm_threshold_management_write_int : INT ;
{attribute 'ac_persist' := 'PersistenceChannel'}
Low_temperature_alarm_threshold : REAL ;
{attribute 'ac_persist' := 'PersistenceChannel'}
High_temperature_alarm_threshold : REAL ;
Low_temperature_alarm_thres_write  : REAL := -20.0 ;
High_temperature_alarm_thres_write : REAL := 20.0 ;
Low_temperature_alarm_thres_write_word : WORD ;
High_temperature_alarm_thres_write_word : WORD ;
muteAlarm : WORD := 1;

{attribute 'ac_persist' := 'PersistenceChannel'}
Low_temperature_alarm_differential : REAL ;
{attribute 'ac_persist' := 'PersistenceChannel'}
High_temperature_alarm_differential : REAL ;
{attribute 'ac_persist' := 'PersistenceChannel'}
Probe_used_for_temperature_alarm_detection : REAL ;
{attribute 'ac_persist' := 'PersistenceChannel'}
Temperature_alarm_delay : REAL ;
Temperature_alarm_delay_write_int : INT ;
{attribute 'ac_persist' := 'PersistenceChannel'}
Operation_in_case_of_high_condenser_alarm : REAL ;
{attribute 'ac_persist' := 'PersistenceChannel'}
Condensation_temperature_alarm : REAL ;
{attribute 'ac_persist' := 'PersistenceChannel'}
Standby_button_enabling : REAL ;
{attribute 'ac_persist' := 'PersistenceChannel'}
Door_switch_input_mode : REAL ;
Door_switch_input_mode_write_int : INT ;
{attribute 'ac_persist' := 'PersistenceChannel'}
Door_alarm_delay : REAL ;
Door_alarm_delay_write_int : INT ;
{attribute 'ac_persist' := 'PersistenceChannel'}
Compressor_stop_delay : REAL ;
Compressor_stop_delay_write_int : INT ;
{attribute 'ac_persist' := 'PersistenceChannel'}
Door_stop_timeout : REAL ;
Door_stop_timeout_write_int : INT ;
{attribute 'ac_persist' := 'PersistenceChannel'}
DI1_digital_input_operation : REAL ;
{attribute 'ac_persist' := 'PersistenceChannel'}
DI1_digital_input_activation : REAL ;
{attribute 'ac_persist' := 'PersistenceChannel'}
DI2_digital_input_operation : REAL ;
{attribute 'ac_persist' := 'PersistenceChannel'}
DI2_digital_input_activation : REAL ;
DI1_digital_input_operation_write_int : INT ;
DI1_digital_input_activation_write_int : INT ;
DI2_digital_input_operation_write_int : INT ;
DI2_digital_input_activation_write_int : INT ;
{attribute 'ac_persist' := 'PersistenceChannel'}
Light_control_mode : REAL ;
Light_control_mode_write_int : INT ;
{attribute 'ac_persist' := 'PersistenceChannel'}
standby : REAL;
standby_write : INT;
{attribute 'ac_persist' := 'PersistenceChannel'}
Light_control : REAL;

write_data_alarm : R_TRIG;
write_data_setp : R_TRIG;
write_data_defrost : R_TRIG;
write_data_mute : R_TRIG;
write_data_control : R_TRIG;
write_data_man_defrost : R_TRIG;
door_open_trigger : R_TRIG ;
door_close_trigger : F_TRIG ;
set_param_trigger : R_TRIG ;
get_param_trigger : R_TRIG ;
all_param_read : BOOL ;
no_loop : INT :=0 ;


control_button : BOOL  := TRUE ;
defrost_button : BOOL  := FALSE ;
setpoint_button : BOOL ;
read_param_button : BOOL ;
{attribute 'ac_persist' := 'PersistenceChannel'}
RL1_output_operation : REAL ;
{attribute 'ac_persist' := 'PersistenceChannel'}
RL2_output_operation : REAL ;
{attribute 'ac_persist' := 'PersistenceChannel'}
RL3_output_operation : REAL ;
{attribute 'ac_persist' := 'PersistenceChannel'}
RL4_output_operation : REAL ;
RL1_output_operation_write_int : INT ;
RL2_output_operation_write_int : INT ;
RL3_output_operation_write_int : INT ;
RL4_output_operation_write_int : INT ;
{attribute 'ac_persist' := 'PersistenceChannel'}
Probe_T1_offset : REAL ;
{attribute 'ac_persist' := 'PersistenceChannel'}
Probe_T2_enable : REAL ;
{attribute 'ac_persist' := 'PersistenceChannel'}
Probe_T2_offset : REAL ;
{attribute 'ac_persist' := 'PersistenceChannel'}
Auxiliary_probe_T3_operation : REAL ;
{attribute 'ac_persist' := 'PersistenceChannel'}
Probe_T3_offset : REAL ;
{attribute 'ac_persist' := 'PersistenceChannel'}
Delay_for_minimum_and_maximum_temperature_logging : REAL ;
{attribute 'ac_persist' := 'PersistenceChannel'}
Selects_the_temperature_probe_to_be_displayed : REAL ;
{attribute 'ac_persist' := 'PersistenceChannel'}
The_relative_weight_of_T2_on_T1 : REAL ;
{attribute 'ac_persist' := 'PersistenceChannel'}
Display_slowdown : REAL ;
Display_slowdown_write_int : INT ;
{attribute 'ac_persist' := 'PersistenceChannel'}
Address_for_PC_communication : REAL ;
Address_for_PC_communication_write_int : INT ;
{attribute 'ac_persist' := 'PersistenceChannel'}
Modbus_protocol_selection : REAL ;
Modbus_protocol_selection_write_int : INT ;
// Word variables
Status_BITs_0_to_15 : WORD;
Status_BITs_16_to_31 : WORD;
Alarm_BITs_0_to_15 : WORD;
setp_write_word : WORD ;
Fan_stop_temperature_write_word : WORD ;

dig1 : BOOL;
dig2 : BOOL;
dout1 : BOOL;
dout2 : BOOL;
dout3 : BOOL;
dout4 : BOOL;
alarm : BOOL;
buzzer_mute : BOOL;
defrost : BOOL;
door_open : BOOL;
test : BOOL;
machine_standby : BOOL;
T1_failure  : BOOL;
T2_failure  : BOOL;
T3_failure  : BOOL;
Low_temperature  : BOOL;
High_temperature  : BOOL;
High_condenser_temperature  : BOOL;
Generic_alarm  : BOOL;
Door_open_alarm  : BOOL;
RL1 : BOOL;
RL2 : BOOL;
RL3 : BOOL;
SSR : BOOL;
deactivate_defrost_button : BOOL ;
modbus_communication : BOOL ;
comm_indicator : REAL ;



//triggers for writing setpoints and parameters
xtrigger_alarm : BOOL;
xtrigger_setp : BOOL;
xtrigger_defrost : BOOL;
xtrigger_mute : BOOL;
xtrigger_control : BOOL;
xtrigger_man_defrost : BOOL;
xtrigger_get_param : BOOL;
xtrigger_set_param : BOOL;







//Graphic variables
Unit_switch_status : INT;
i : INT;
show_trendvalue : ARRAY[0..50] OF BOOL;
select_trendvalue : INT :=0 ;

END_VAR




temp_provision_room:= scaleFunction(modbus_var[0],0.1, 0);
temp_defrost := scaleFunction(modbus_var[1],0.1, 0);
reg2 := scaleFunction(modbus_var[2],0.1, 0); // not used ?
reg3 := scaleFunction(modbus_var[3],0.1, 0); // not used ?
reg4 := scaleFunction(modbus_var[4],0.1, 0); // not used ?
reg5 := scaleFunction(modbus_var[5],0.1, 0); // not used ?
reg6 := scaleFunction(modbus_var[6],0.1, 0); // not used ?
reg7 := scaleFunction(modbus_var[7],0.1, 0); // not used ?
reg8 := scaleFunction(modbus_var[8],0.1, 0); // not used ?
reg9 := scaleFunction(modbus_var[9],0.1, 0); // not used ?
reg10 := modbus_var[10]; // not used ?
set_point := scaleFunction(modbus_var[11],0.1, 0);  // not used ?
reg12 := scaleFunction(modbus_var[12],0.1, 0); // not used ?
reg13 := scaleFunction(modbus_var[13],0.1, 0); // not used ?
reg14 := scaleFunction(modbus_var[14],0.1, 0); // not used ?
reg15 := scaleFunction(modbus_var[15],0.1, 0); // not used ?
reg16 := scaleFunction(modbus_var[16],0.1, 0); // not used ?
reg17 := scaleFunction(modbus_var[17],0.1, 0); // not used ?

// Non changeable parameters

T1_offset := scaleFunction(modbus_var1[2000],1, 0);
T2_offset := scaleFunction(modbus_var1[2001],1, 2);
T3_offset := scaleFunction(modbus_var1[2002],1, 3);
T1_span := scaleFunction(modbus_var1[2003],1, 4);
T2_span := scaleFunction(modbus_var1[2004],1, 5);
T3_span := scaleFunction(modbus_var1[2005],1, 6);

valore_tasto1_V := scaleFunction(modbus_var[150],1, 6);
valore_tasto_UP := scaleFunction(modbus_var[151],1, 6);
valore_tasto_DW := scaleFunction(modbus_var[152],1, 6);
valore_tasto_X := scaleFunction(modbus_var[153],1, 6);

Test_display := scaleFunction(modbus_var[193],1, 0);
Tasto_attualmente_premuto := scaleFunction(modbus_var[194],1, 0);
Password := scaleFunction(modbus_var[197],1, 0);

preset_parameters:= scaleFunction(modbus_var[200],1, 0);

Setpoint:= scaleFunction(modbus_var[303],0.1, 0);
Thermostat_OFF_ON_ref_to_SP:= scaleFunction(modbus_var[304],0.1, 0);
Thermostat_ON_OFF_ref_to_SP:= scaleFunction(modbus_var[305],0.1, 0);

Defrost_start_mode:= scaleFunction(modbus_var[400],1, 0);
Time_based_defrost:= scaleFunction(modbus_var[401],1, 0);

Delay_for_pressure_equalization_for_hot_gas:= scaleFunction(modbus_var[405],1, 0);

Defrost_end_temperature:= scaleFunction(modbus_var[406],0.1, 0);
Maximum_defrost_duration:= scaleFunction(modbus_var[407],1, 0);

Drain_down_time:= scaleFunction(modbus_var[408],1, 0);
Display_defrost_mode:= scaleFunction(modbus_var[409],1, 0);

Target_evaporator_temperature:= scaleFunction(modbus_var[453],0.1, 0);
Fan_stop_delay_after_compressor_stop:= scaleFunction(modbus_var[454],1, 0);
Timed_fan_stop:= scaleFunction(modbus_var[455],1, 0);
Timed_fan_run:= scaleFunction(modbus_var[456],1, 0);
Fan_Minimum_Stop:= scaleFunction(modbus_var[457],1, 0);


Low_temperature_alarm_threshold:= scaleFunction(modbus_var[501],0.1, 0);
High_temperature_alarm_threshold:= scaleFunction(modbus_var[502],0.1, 0);
Low_temperature_alarm_differential:= scaleFunction(modbus_var[503],0.1, 0);
High_temperature_alarm_differential:= scaleFunction(modbus_var[504],0.1, 0);
Probe_used_for_temperature_alarm_detection:= scaleFunction(modbus_var[505],1, 0);
Operation_in_case_of_high_condenser_alarm:= scaleFunction(modbus_var[507],1, 0);
Condensation_temperature_alarm:= scaleFunction(modbus_var[508],0.1, 0);

Standby_button_enabling:= scaleFunction(modbus_var[600],1, 0);



// Changeable parameters
delay_timer(IN:=read_param_button, PT:=set_delaytime);
IF read_param_button THEN
	Display_slowdown:= scaleFunction(modbus_var[208],1, 0);
	Readout_scale:= scaleFunction(modbus_var[300],1, 0);
	Minimum_temperature_setpoint:= scaleFunction(modbus_var[301],0.1, 0);
	Maximum_temperature_setpoint:= scaleFunction(modbus_var[302],0.1, 0);
	CH_minimum_OFF_time:= scaleFunction(modbus_var[306],1, 0);
	CH_minimum_ON_time:= scaleFunction(modbus_var[307],1, 0);
	CH_output_ON_when_probe_T1_is_faulty:= scaleFunction(modbus_var[308],1, 0);
	CH_output_OFF_when_probe_T1_is_faulty:= scaleFunction(modbus_var[309],1, 0);
	Minimum_Time_Between_Defrost:= scaleFunction(modbus_var[402],1, 0);
	Defrost_time_optimization:= scaleFunction(modbus_var[403],1, 0);
	Defrost_type:= scaleFunction(modbus_var[404],1, 0);
//	Defrost_end_temperature:= scaleFunction(modbus_var[406],1, 0);
//	Maximum_defrost_duration:= scaleFunction(modbus_var[407],1, 0);
	Display_delay:= scaleFunction(modbus_var[410],1, 0);
	Fans_active_during_defrost:= scaleFunction(modbus_var[411],1, 0);
	Fan_restart_temperature_after_defrost:= scaleFunction(modbus_var[412],0.1, 0);
	Fan_mode_during_thermostatic_control:= scaleFunction(modbus_var[452],1, 0);
	Fan_stop_temperature:= scaleFunction(modbus_var[450],0.1, 0);
	Maximum_fan_stop_for_FDD_FET:= scaleFunction(modbus_var[451],1, 0);
	Alarm_threshold_management:= scaleFunction(modbus_var[500],1, 0);
	Temperature_alarm_delay:= scaleFunction(modbus_var[506],1, 0);
	Door_switch_input_mode:= scaleFunction(modbus_var[601],1, 0);
	Door_alarm_delay:= scaleFunction(modbus_var[602],1, 0);
	Compressor_stop_delay:= scaleFunction(modbus_var[603],1, 0);
	Door_stop_timeout:= scaleFunction(modbus_var[604],1, 0);
	DI1_digital_input_operation:= scaleFunction(modbus_var[605],1, 0);
	DI1_digital_input_activation:= scaleFunction(modbus_var[606],1, 0);
	DI2_digital_input_operation:= scaleFunction(modbus_var[607],1, 0);
	DI2_digital_input_activation:= scaleFunction(modbus_var[608],1, 0);
	Light_control_mode:= scaleFunction(modbus_var[609],1, 0);
	RL1_output_operation:= scaleFunction(modbus_var[650],1, 0);
	RL2_output_operation:= scaleFunction(modbus_var[651],1, 0);
	RL3_output_operation:= scaleFunction(modbus_var[652],1, 0);
	RL4_output_operation:= scaleFunction(modbus_var[653],1, 0);

	// no_loop :=no_loop +1 ;
	IF delay_timer.Q THEN
		read_param_button := FALSE ;
		no_loop:=0;
	END_IF	
END_IF










standby:= scaleFunction(modbus_var[702],1, 0);
Light_control:= scaleFunction(modbus_var[703],1, 0);




Probe_T1_offset:= scaleFunction(modbus_var[201],0.1, 0);
Probe_T2_enable:= scaleFunction(modbus_var[202],1, 0);
Probe_T2_offset:= scaleFunction(modbus_var[203],0.1, 0);
Auxiliary_probe_T3_operation:= scaleFunction(modbus_var[204],1, 0);
Probe_T3_offset:= scaleFunction(modbus_var[205],0.1, 0);
Selects_the_temperature_probe_to_be_displayed:= scaleFunction(modbus_var[206],1, 0);
The_relative_weight_of_T2_on_T1:= scaleFunction(modbus_var[207],1, 0);

Address_for_PC_communication:= scaleFunction(modbus_var[209],1, 0);
Modbus_protocol_selection:= scaleFunction(modbus_var[210],1, 0);
Delay_for_minimum_and_maximum_temperature_logging:= scaleFunction(modbus_var[211],1, 0);

//  Statusbits
Status_BITs_0_to_15 := modbus_var[100];
Status_BITs_16_to_31 := modbus_var[102];
Alarm_BITs_0_to_15 := modbus_var[101];


alarm := maskbitFunction(Status_BITs_0_to_15,0) OR NOT modbus_communication ;
buzzer_mute := maskbitFunction(Status_BITs_0_to_15,1);
defrost:= maskbitFunction(Status_BITs_0_to_15,2);
door_open := maskbitFunction(Status_BITs_0_to_15,3);
test := maskbitFunction(Status_BITs_0_to_15,4);
machine_standby := maskbitFunction(Status_BITs_0_to_15,5);


T1_failure := maskbitFunction(Alarm_BITs_0_to_15,0);
T2_failure := maskbitFunction(Alarm_BITs_0_to_15,1);
T3_failure := maskbitFunction(Alarm_BITs_0_to_15,2);
Low_temperature := maskbitFunction(Alarm_BITs_0_to_15,3);
High_temperature := maskbitFunction(Alarm_BITs_0_to_15,4);
High_condenser_temperature := maskbitFunction(Alarm_BITs_0_to_15,5);
Generic_alarm := maskbitFunction(Alarm_BITs_0_to_15,6);
Door_open_alarm := maskbitFunction(Alarm_BITs_0_to_15,7);

dout1 := maskbitFunction(Status_BITs_16_to_31,0); 
dout2 := maskbitFunction(Status_BITs_16_to_31,1);
dout3 := maskbitFunction(Status_BITs_16_to_31,2);
dout4 := maskbitFunction(Status_BITs_16_to_31,3);

RL1 := maskbitFunction(modbus_var[196],0);
RL2 := maskbitFunction(modbus_var[196],1);

RL3 := maskbitFunction(modbus_var[196],2);
SSR := maskbitFunction(modbus_var[196],3);


dig1 := maskbitFunction(reg10,0);
dig2 := maskbitFunction(reg10,1);

// Communication fault
comm_indicator := temp_provision_room + temp_defrost + reg2 + reg3 + reg4 + reg5
+ reg6 + reg7 + reg8 + reg9 + reg10 ;
IF comm_indicator = 0 THEN
	modbus_communication := FALSE ;
ELSE
	modbus_communication := TRUE ;
END_IF
	



// Parameter write values

setp_write_word := REAL_TO_INT(setp_write*10) ;
Thermostat_OFF_ON_write_word := REAL_TO_INT(Thermostat_OFF_ON_write*10) ;
Thermostat_ON_OFF_write_word:= REAL_TO_INT(Thermostat_ON_OFF_write*10) ;
Low_temperature_alarm_thres_write_word:= REAL_TO_INT(Low_temperature_alarm_thres_write*10);
High_temperature_alarm_thres_write_word:= REAL_TO_INT(High_temperature_alarm_thres_write*10);
muteAlarm :=1 ;
Time_based_defrost_write_word:= REAL_TO_INT(Time_based_defrost_write*1);
Defrost_end_temperature_write_word:= REAL_TO_INT(Defrost_end_temperature_write*10);
Drain_down_time_write_int:= REAL_TO_INT(Drain_down_time_write);
Maximum_defrost_duration_write_word:= REAL_TO_INT(Maximum_defrost_duration_write*1);
Fan_stop_temperature_write_word:= REAL_TO_INT(Fan_stop_temperature*10);
preset_parameters_write_int:=REAL_TO_INT(preset_parameters);
Readout_scale_write_int:=REAL_TO_INT(Readout_scale);
Minimum_temperature_setpoint_write_int:=REAL_TO_INT(Minimum_temperature_setpoint*10);
Maximum_temperature_setpoint_write_int:=REAL_TO_INT(Maximum_temperature_setpoint*10);
CH_minimum_OFF_time_write_int:=REAL_TO_INT(CH_minimum_OFF_time);
CH_minimum_ON_time_write_int:=REAL_TO_INT(CH_minimum_ON_time);
CH_output_ON_when_probe_T1_is_faulty_write_int:=REAL_TO_INT(CH_output_ON_when_probe_T1_is_faulty);
CH_output_OFF_when_probe_T1_is_faulty_write_int:=REAL_TO_INT(CH_output_OFF_when_probe_T1_is_faulty);
Minimum_Time_Between_Defrost_write_int:=REAL_TO_INT(Minimum_Time_Between_Defrost);
Defrost_time_optimization_write_int:=REAL_TO_INT(Defrost_time_optimization);
Defrost_type_write_int:=REAL_TO_INT(Defrost_type);
Display_delay_write_int:=REAL_TO_INT(Display_delay);
Fans_active_during_defrost_write_int:=REAL_TO_INT(Fans_active_during_defrost);
Fan_restart_temperature_after_defrost_write_int:=REAL_TO_INT(Fan_restart_temperature_after_defrost*10);
// Fan_stop_temperature_write_int:=REAL_TO_INT(Fan_stop_temperature);
Maximum_fan_stop_for_FDD_FET_write_int:=REAL_TO_INT(Maximum_fan_stop_for_FDD_FET);
Fan_mode_during_thermostatic_control_write_int:=REAL_TO_INT(Fan_mode_during_thermostatic_control);
Alarm_threshold_management_write_int:=REAL_TO_INT(Alarm_threshold_management);
Temperature_alarm_delay_write_int:=REAL_TO_INT(Temperature_alarm_delay);
Door_switch_input_mode_write_int:=REAL_TO_INT(Door_switch_input_mode);
Door_alarm_delay_write_int:=REAL_TO_INT(Door_alarm_delay);
Compressor_stop_delay_write_int:=REAL_TO_INT(Compressor_stop_delay);
Door_stop_timeout_write_int:=REAL_TO_INT(Door_stop_timeout);
DI1_digital_input_operation_write_int:=REAL_TO_INT(DI1_digital_input_operation);
DI1_digital_input_activation_write_int:=REAL_TO_INT(DI1_digital_input_activation);
DI2_digital_input_operation_write_int:=REAL_TO_INT(DI2_digital_input_operation);
DI2_digital_input_activation_write_int:=REAL_TO_INT(DI2_digital_input_activation);
Light_control_mode_write_int:=REAL_TO_INT(Light_control_mode);
RL1_output_operation_write_int:=REAL_TO_INT(RL1_output_operation);
RL2_output_operation_write_int:=REAL_TO_INT(RL2_output_operation);
RL3_output_operation_write_int:=REAL_TO_INT(RL3_output_operation);
RL4_output_operation_write_int:=REAL_TO_INT(RL4_output_operation);
Display_slowdown_write_int:=REAL_TO_INT(Display_slowdown);
Address_for_PC_communication_write_int:=REAL_TO_INT(Address_for_PC_communication);
Modbus_protocol_selection_write_int:=REAL_TO_INT(Modbus_protocol_selection);

write_data_alarm(clk:=xtrigger_alarm);
write_data_setp(clk:=xtrigger_setp);
write_data_defrost(clk:=xtrigger_defrost);
write_data_mute(clk:=xtrigger_mute);
write_data_control(clk:=xtrigger_control);
write_data_man_defrost(clk:=xtrigger_man_defrost);
get_param_trigger(clk:=xtrigger_get_param);
set_param_trigger(clk:=xtrigger_set_param);


IF control_button THEN
	standby_write := 0 ;
	IF machine_standby=TRUE THEN
		xtrigger_control := TRUE;
	END_IF
ELSE
	standby_write := 1 ;
	IF machine_standby=FALSE THEN
		xtrigger_control := TRUE;
	END_IF	
END_IF


IF defrost_button THEN
	defrost_write := 1 ;
	IF defrost=FALSE THEN
		xtrigger_man_defrost := TRUE;
	END_IF
ELSE
	defrost_write := 0 ;

END_IF

// Door open timers
door_open_trigger(clk:=door_open);
door_close_trigger(clk:=door_open);

timer_door_open(IN:=timer_enable, PT:=T#30D);
timer_door_closed(IN:=timer2_enable, PT:=T#30D);

IF door_open_trigger.Q THEN
	closetime_tot := opentime_tot + timer_door_closed.ET;
	timer_enable := TRUE;
	timer2_enable := FALSE;
END_IF

IF door_close_trigger.Q THEN
	opentime_tot := opentime_tot + timer_door_open.ET;
	timer_enable := FALSE;
	timer2_enable := TRUE ;
END_IF


total_time := opentime_tot + closetime_tot ;

opentime_ms := TO_LREAL(TO_UDINT(opentime_tot) / 1000.0);
totaltime_ms := TO_LREAL(TO_UDINT(total_time) / 1000.0);

opentime_proc := (opentime_ms /totaltime_ms)*100 ;
IF resettimer_button THEN
	opentime_tot := T#0S ;
	closetime_tot := T#0S ;
	total_time := T#0S;
END_IF






// Graphic controls
IF select_trendvalue > 0 THEN
	show_trendvalue[select_trendvalue]:= TRUE;
ELSIF select_trendvalue = 0 THEN
	FOR i := 0 TO 50 DO
      show_trendvalue[i] := FALSE;
   	END_FOR
END_IF ;

END_PROGRAM

// Device/Application/Provision_2
PROGRAM Provision_2
VAR




modbus_var : ARRAY[0..800] OF WORD;
modbus_var1 : ARRAY[2000..2010] OF WORD;
timer_door_open : TON ;
timer_door_closed : TON ;
delay_timer : TON ;
open_time : TIME ;
total_time : TIME ;
opentime_tot : TIME ;
opentime_proc : REAL ;
closetime_tot : TIME ; 
{attribute 'ac_persist' := 'PersistenceChannel'}
set_delaytime : TIME := T#1S;
timer_enable : BOOL;
timer2_enable : BOOL;
timer_elapsed : BOOL ;
start_timer : BOOL := TRUE;
doorclose : F_TRIG;
resettimer_button :BOOL ;
totaltime_ms : LREAL ;
opentime_ms : LREAL ;

temp_provision_room : REAL;
temp_defrost : REAL;
regulator_temp : REAL;

set_point: REAL;
reg2 : REAL ;
reg3 : REAL ;
reg4 : REAL ;
reg5 : REAL ;
reg6 : REAL ;
reg7 : REAL ;
reg8 : REAL ;
reg9 : REAL ;
reg10 : WORD ;
reg11 : REAL ;
reg12 : REAL ;
reg13 : REAL ;
reg14 : REAL ;
reg15 : REAL ;
reg16 : REAL ;
reg17 : REAL ;
T1_offset : REAL ;
T2_offset : REAL ;
T3_offset : REAL ;
T1_span : REAL ;
T2_span : REAL ;
T3_span : REAL ;
valore_tasto1_V : REAL ;
valore_tasto_UP : REAL ;
valore_tasto_DW : REAL ;
valore_tasto_X : REAL ;
Test_display : REAL ;
Tasto_attualmente_premuto : REAL ;
Password : REAL ;

{attribute 'ac_persist' := 'PersistenceChannel'}
preset_parameters : REAL ;
preset_parameters_write_int :INT;
{attribute 'ac_persist' := 'PersistenceChannel'}
Readout_scale : REAL ;
{attribute 'ac_persist' := 'PersistenceChannel'}
Readout_scale_write_int : INT;
{attribute 'ac_persist' := 'PersistenceChannel'}
Minimum_temperature_setpoint : REAL ;
Minimum_temperature_setpoint_write_int : INT ;
{attribute 'ac_persist' := 'PersistenceChannel'}
Maximum_temperature_setpoint : REAL ;
Maximum_temperature_setpoint_write_int : INT ;
setp_write : REAL ;
{attribute 'ac_persist' := 'PersistenceChannel'}
Setpoint : REAL ;
{attribute 'ac_persist' := 'PersistenceChannel'}
Thermostat_OFF_ON_ref_to_SP : REAL  ;
{attribute 'ac_persist' := 'PersistenceChannel'}
Thermostat_ON_OFF_ref_to_SP : REAL  ;
Thermostat_OFF_ON_write : REAL  := 1.0 ;
Thermostat_ON_OFF_write : REAL  := 1.0 ;
Thermostat_OFF_ON_write_word : WORD ;
Thermostat_ON_OFF_write_word : WORD ;
Time_based_defrost_write : REAL   := 8.0  ;
Time_based_defrost_write_word : WORD  ;
Defrost_end_temperature_write : REAL  := 20.0 ;
Defrost_end_temperature_write_word : WORD ;
Fan_restart_temperature_after_defrost_write : REAL ;
Fan_restart_temperature_after_defrost_write_int : INT ;
Maximum_defrost_duration_write : REAL ;
Maximum_defrost_duration_write_word : WORD ;
defrost_write : WORD :=0 ;
{attribute 'ac_persist' := 'PersistenceChannel'}
CH_minimum_OFF_time : REAL ;
CH_minimum_OFF_time_write_int : INT ;
{attribute 'ac_persist' := 'PersistenceChannel'}
CH_minimum_ON_time : REAL ;
CH_minimum_ON_time_write_int : INT ;
{attribute 'ac_persist' := 'PersistenceChannel'}
CH_output_ON_when_probe_T1_is_faulty : REAL ;
CH_output_ON_when_probe_T1_is_faulty_write_int : INT ;
{attribute 'ac_persist' := 'PersistenceChannel'}
CH_output_OFF_when_probe_T1_is_faulty : REAL ;
CH_output_OFF_when_probe_T1_is_faulty_write_int : INT ;

{attribute 'ac_persist' := 'PersistenceChannel'}
Defrost_start_mode : REAL ;
{attribute 'ac_persist' := 'PersistenceChannel'}
Time_based_defrost : REAL ;
{attribute 'ac_persist' := 'PersistenceChannel'}
Minimum_Time_Between_Defrost : REAL ;
Minimum_Time_Between_Defrost_write_int : INT;
{attribute 'ac_persist' := 'PersistenceChannel'}
Defrost_time_optimization : REAL ;
Defrost_time_optimization_write_int : INT;
{attribute 'ac_persist' := 'PersistenceChannel'}
Defrost_type : REAL ;
Defrost_type_write_int : INT;
{attribute 'ac_persist' := 'PersistenceChannel'}
Delay_for_pressure_equalization_for_hot_gas : REAL ;
{attribute 'ac_persist' := 'PersistenceChannel'}
Defrost_end_temperature : REAL ;
{attribute 'ac_persist' := 'PersistenceChannel'}
Maximum_defrost_duration : REAL ;
{attribute 'ac_persist' := 'PersistenceChannel'}
Drain_down_time : REAL ;
Drain_down_time_write : REAL;
Drain_down_time_write_int : INT;
{attribute 'ac_persist' := 'PersistenceChannel'}
Display_defrost_mode : REAL ;
{attribute 'ac_persist' := 'PersistenceChannel'}
Display_delay : REAL ;
Display_delay_write_int : INT;
{attribute 'ac_persist' := 'PersistenceChannel'}
Fans_active_during_defrost : REAL ;
Fans_active_during_defrost_write_int : INT;
{attribute 'ac_persist' := 'PersistenceChannel'}
Fan_restart_temperature_after_defrost : REAL ;
{attribute 'ac_persist' := 'PersistenceChannel'}
Fan_stop_temperature : REAL ;
Fan_stop_temperature_write_int : INT ;
{attribute 'ac_persist' := 'PersistenceChannel'}
Maximum_fan_stop_for_FDD_FET : REAL ;
Maximum_fan_stop_for_FDD_FET_write_int : INT ;
{attribute 'ac_persist' := 'PersistenceChannel'}
Fan_mode_during_thermostatic_control : REAL ;
Fan_mode_during_thermostatic_control_write_int : INT ;
{attribute 'ac_persist' := 'PersistenceChannel'}
Target_evaporator_temperature : REAL ;
{attribute 'ac_persist' := 'PersistenceChannel'}
Fan_stop_delay_after_compressor_stop : REAL ;
{attribute 'ac_persist' := 'PersistenceChannel'}
Timed_fan_stop : REAL ;
{attribute 'ac_persist' := 'PersistenceChannel'}
Timed_fan_run : REAL ;
{attribute 'ac_persist' := 'PersistenceChannel'}
Fan_Minimum_Stop : REAL ;
{attribute 'ac_persist' := 'PersistenceChannel'}
Alarm_threshold_management : REAL ;
Alarm_threshold_management_write_int : INT ;
{attribute 'ac_persist' := 'PersistenceChannel'}
Low_temperature_alarm_threshold : REAL ;
{attribute 'ac_persist' := 'PersistenceChannel'}
High_temperature_alarm_threshold : REAL ;
Low_temperature_alarm_thres_write  : REAL := -20.0 ;
High_temperature_alarm_thres_write : REAL := 20.0 ;
Low_temperature_alarm_thres_write_word : WORD ;
High_temperature_alarm_thres_write_word : WORD ;
muteAlarm : WORD := 1;

